REGION Network 5: Клапан регулирующий - 5
   // Зона 7
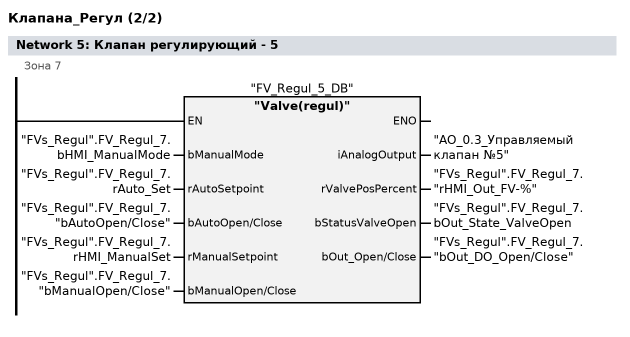
   RUNG wire#powerrail
      "FV_Regul_5_DB"(bManualMode := "FVs_Regul".FV_Regul_7.bHMI_ManualMode, rAutoSetpoint := "FVs_Regul".FV_Regul_7.rAuto_Set, "bAutoOpen/Close" := "FVs_Regul".FV_Regul_7."bAutoOpen/Close", rManualSetpoint := "FVs_Regul".FV_Regul_7.rHMI_ManualSet, "bManualOpen/Close" := "FVs_Regul".FV_Regul_7."bManualOpen/Close", iAnalogOutput => "AO_0.3_Управляемый клапан №5", rValvePosPercent => "FVs_Regul".FV_Regul_7."rHMI_Out_FV-%", bStatusValveOpen => "FVs_Regul".FV_Regul_7.bOut_State_ValveOpen, "bOut_Open/Close" => "FVs_Regul".FV_Regul_7."bOut_DO_Open/Close")
   END_RUNG
   // the same network as SCL:
   "FV_Regul_5_DB"(bManualMode := "FVs_Regul".FV_Regul_7.bHMI_ManualMode,   // "Valve(regul)"
                   rAutoSetpoint := "FVs_Regul".FV_Regul_7.rAuto_Set,
                   "bAutoOpen/Close" := "FVs_Regul".FV_Regul_7."bAutoOpen/Close",
                   rManualSetpoint := "FVs_Regul".FV_Regul_7.rHMI_ManualSet,
                   "bManualOpen/Close" := "FVs_Regul".FV_Regul_7."bManualOpen/Close",
                   iAnalogOutput => "AO_0.3_Управляемый клапан №5",
                   rValvePosPercent => "FVs_Regul".FV_Regul_7."rHMI_Out_FV-%",
                   bStatusValveOpen => "FVs_Regul".FV_Regul_7.bOut_State_ValveOpen,
                   "bOut_Open/Close" => "FVs_Regul".FV_Regul_7."bOut_DO_Open/Close");
END_REGION

REGION Network 6 (SCL): Клапана регулирующие ручной режим с вфходом DO
   // Для перевода клапана регулирующего в ручной режим должен перейти по сигналу от ручного режим с клапана DO, т.е. для работы клапана регулирующего необходим сигнал DO
   (*"FVs_o/p".FV_1.bManualMode := "FVs_Regul".FV_Regul_1.bHMI_ManualMode;
   "FVs_o/p".FV_2.bManualMode := "FVs_Regul".FV_Regul_2.bHMI_ManualMode;
   "FVs_o/p".FV_3.bManualMode := "FVs_Regul".FV_Regul_3.bHMI_ManualMode;
   "FVs_o/p".FV_4.bManualMode := "FVs_Regul".FV_Regul_5.bHMI_ManualMode;
   *)
END_REGION
END_FUNCTION

FUNCTION "Зоны пастеризации_Контроль" : Void   // FC3, LAD
{ S7_Optimized_Access := 'TRUE' }
VERSION : 0.1
BEGIN

REGION Network 1: Зона 1
   // Зона 1
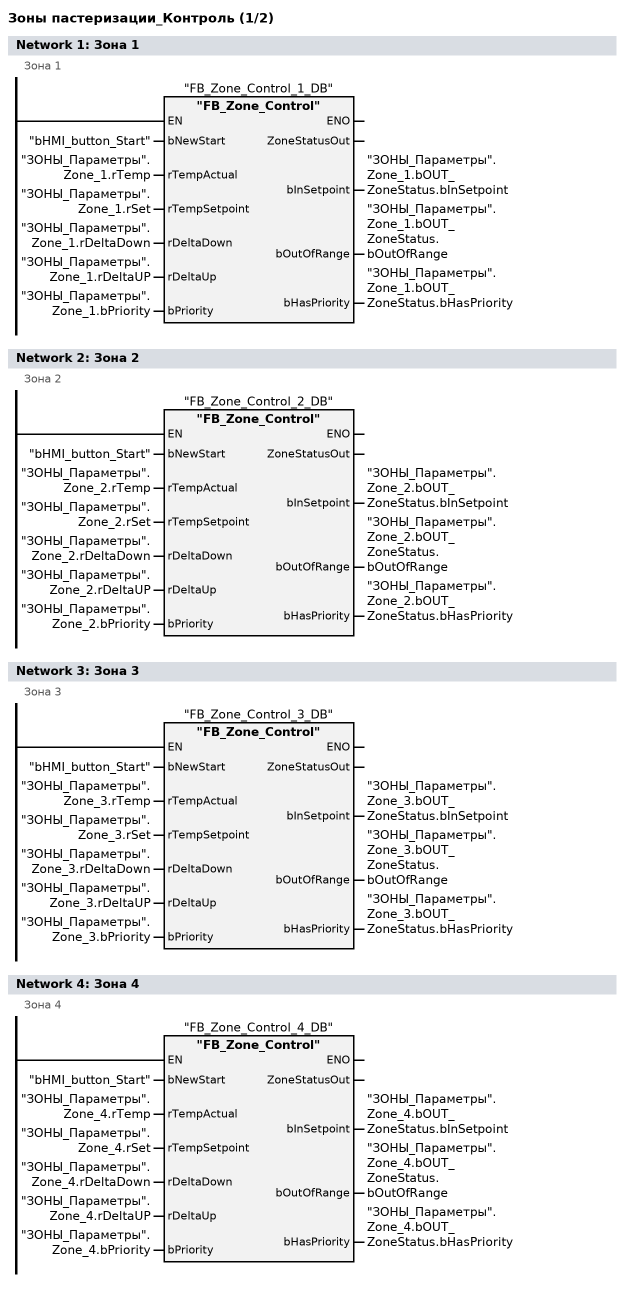
   RUNG wire#powerrail
      "FB_Zone_Control_1_DB"(bNewStart := "bHMI_button_Start", rTempActual := "ЗОНЫ_Параметры".Zone_1.rTemp, rTempSetpoint := "ЗОНЫ_Параметры".Zone_1.rSet, rDeltaDown := "ЗОНЫ_Параметры".Zone_1.rDeltaDown, rDeltaUp := "ЗОНЫ_Параметры".Zone_1.rDeltaUP, bPriority := "ЗОНЫ_Параметры".Zone_1.bPriority, ZoneStatusOut =>, bInSetpoint => "ЗОНЫ_Параметры".Zone_1.bOUT_ZoneStatus.bInSetpoint, bOutOfRange => "ЗОНЫ_Параметры".Zone_1.bOUT_ZoneStatus.bOutOfRange, bHasPriority => "ЗОНЫ_Параметры".Zone_1.bOUT_ZoneStatus.bHasPriority)
   END_RUNG
   // the same network as SCL:
   "FB_Zone_Control_1_DB"(bNewStart := "bHMI_button_Start",   // "FB_Zone_Control"
                          rTempActual := "ЗОНЫ_Параметры".Zone_1.rTemp,
                          rTempSetpoint := "ЗОНЫ_Параметры".Zone_1.rSet,
                          rDeltaDown := "ЗОНЫ_Параметры".Zone_1.rDeltaDown,
                          rDeltaUp := "ЗОНЫ_Параметры".Zone_1.rDeltaUP,
                          bPriority := "ЗОНЫ_Параметры".Zone_1.bPriority,
                          bInSetpoint => "ЗОНЫ_Параметры".Zone_1.bOUT_ZoneStatus.bInSetpoint,
                          bOutOfRange => "ЗОНЫ_Параметры".Zone_1.bOUT_ZoneStatus.bOutOfRange,
                          bHasPriority => "ЗОНЫ_Параметры".Zone_1.bOUT_ZoneStatus.bHasPriority);
END_REGION

REGION Network 2: Зона 2
   // Зона 2
   RUNG wire#powerrail
      "FB_Zone_Control_2_DB"(bNewStart := "bHMI_button_Start", rTempActual := "ЗОНЫ_Параметры".Zone_2.rTemp, rTempSetpoint := "ЗОНЫ_Параметры".Zone_2.rSet, rDeltaDown := "ЗОНЫ_Параметры".Zone_2.rDeltaDown, rDeltaUp := "ЗОНЫ_Параметры".Zone_2.rDeltaUP, bPriority := "ЗОНЫ_Параметры".Zone_2.bPriority, ZoneStatusOut =>, bInSetpoint => "ЗОНЫ_Параметры".Zone_2.bOUT_ZoneStatus.bInSetpoint, bOutOfRange => "ЗОНЫ_Параметры".Zone_2.bOUT_ZoneStatus.bOutOfRange, bHasPriority => "ЗОНЫ_Параметры".Zone_2.bOUT_ZoneStatus.bHasPriority)
   END_RUNG
   // the same network as SCL:
   "FB_Zone_Control_2_DB"(bNewStart := "bHMI_button_Start",   // "FB_Zone_Control"
                          rTempActual := "ЗОНЫ_Параметры".Zone_2.rTemp,
                          rTempSetpoint := "ЗОНЫ_Параметры".Zone_2.rSet,
                          rDeltaDown := "ЗОНЫ_Параметры".Zone_2.rDeltaDown,
                          rDeltaUp := "ЗОНЫ_Параметры".Zone_2.rDeltaUP,
                          bPriority := "ЗОНЫ_Параметры".Zone_2.bPriority,
                          bInSetpoint => "ЗОНЫ_Параметры".Zone_2.bOUT_ZoneStatus.bInSetpoint,
                          bOutOfRange => "ЗОНЫ_Параметры".Zone_2.bOUT_ZoneStatus.bOutOfRange,
                          bHasPriority => "ЗОНЫ_Параметры".Zone_2.bOUT_ZoneStatus.bHasPriority);
END_REGION

REGION Network 3: Зона 3
   // Зона 3
   RUNG wire#powerrail
      "FB_Zone_Control_3_DB"(bNewStart := "bHMI_button_Start", rTempActual := "ЗОНЫ_Параметры".Zone_3.rTemp, rTempSetpoint := "ЗОНЫ_Параметры".Zone_3.rSet, rDeltaDown := "ЗОНЫ_Параметры".Zone_3.rDeltaDown, rDeltaUp := "ЗОНЫ_Параметры".Zone_3.rDeltaUP, bPriority := "ЗОНЫ_Параметры".Zone_3.bPriority, ZoneStatusOut =>, bInSetpoint => "ЗОНЫ_Параметры".Zone_3.bOUT_ZoneStatus.bInSetpoint, bOutOfRange => "ЗОНЫ_Параметры".Zone_3.bOUT_ZoneStatus.bOutOfRange, bHasPriority => "ЗОНЫ_Параметры".Zone_3.bOUT_ZoneStatus.bHasPriority)
   END_RUNG
   // the same network as SCL:
   "FB_Zone_Control_3_DB"(bNewStart := "bHMI_button_Start",   // "FB_Zone_Control"
                          rTempActual := "ЗОНЫ_Параметры".Zone_3.rTemp,
                          rTempSetpoint := "ЗОНЫ_Параметры".Zone_3.rSet,
                          rDeltaDown := "ЗОНЫ_Параметры".Zone_3.rDeltaDown,
                          rDeltaUp := "ЗОНЫ_Параметры".Zone_3.rDeltaUP,
                          bPriority := "ЗОНЫ_Параметры".Zone_3.bPriority,
                          bInSetpoint => "ЗОНЫ_Параметры".Zone_3.bOUT_ZoneStatus.bInSetpoint,
                          bOutOfRange => "ЗОНЫ_Параметры".Zone_3.bOUT_ZoneStatus.bOutOfRange,
                          bHasPriority => "ЗОНЫ_Параметры".Zone_3.bOUT_ZoneStatus.bHasPriority);
END_REGION

REGION Network 4: Зона 4
   // Зона 4
   RUNG wire#powerrail
      "FB_Zone_Control_4_DB"(bNewStart := "bHMI_button_Start", rTempActual := "ЗОНЫ_Параметры".Zone_4.rTemp, rTempSetpoint := "ЗОНЫ_Параметры".Zone_4.rSet, rDeltaDown := "ЗОНЫ_Параметры".Zone_4.rDeltaDown, rDeltaUp := "ЗОНЫ_Параметры".Zone_4.rDeltaUP, bPriority := "ЗОНЫ_Параметры".Zone_4.bPriority, ZoneStatusOut =>, bInSetpoint => "ЗОНЫ_Параметры".Zone_4.bOUT_ZoneStatus.bInSetpoint, bOutOfRange => "ЗОНЫ_Параметры".Zone_4.bOUT_ZoneStatus.bOutOfRange, bHasPriority => "ЗОНЫ_Параметры".Zone_4.bOUT_ZoneStatus.bHasPriority)
   END_RUNG
   // the same network as SCL:
   "FB_Zone_Control_4_DB"(bNewStart := "bHMI_button_Start",   // "FB_Zone_Control"
                          rTempActual := "ЗОНЫ_Параметры".Zone_4.rTemp,
                          rTempSetpoint := "ЗОНЫ_Параметры".Zone_4.rSet,
                          rDeltaDown := "ЗОНЫ_Параметры".Zone_4.rDeltaDown,
                          rDeltaUp := "ЗОНЫ_Параметры".Zone_4.rDeltaUP,
                          bPriority := "ЗОНЫ_Параметры".Zone_4.bPriority,
                          bInSetpoint => "ЗОНЫ_Параметры".Zone_4.bOUT_ZoneStatus.bInSetpoint,
                          bOutOfRange => "ЗОНЫ_Параметры".Zone_4.bOUT_ZoneStatus.bOutOfRange,
                          bHasPriority => "ЗОНЫ_Параметры".Zone_4.bOUT_ZoneStatus.bHasPriority);
END_REGION

REGION Network 5: Зона 5
   // Зона 5
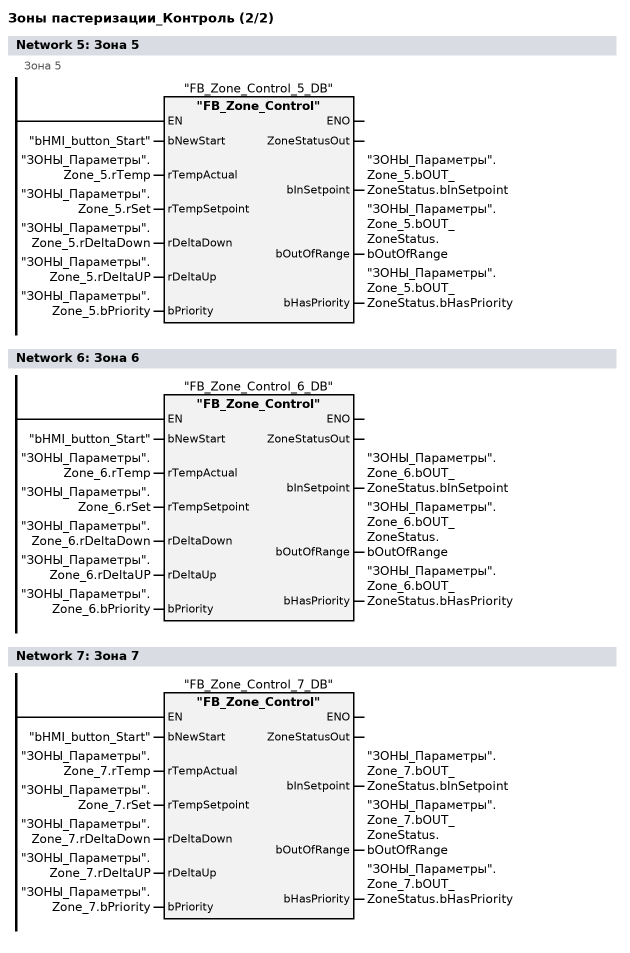
   RUNG wire#powerrail
      "FB_Zone_Control_5_DB"(bNewStart := "bHMI_button_Start", rTempActual := "ЗОНЫ_Параметры".Zone_5.rTemp, rTempSetpoint := "ЗОНЫ_Параметры".Zone_5.rSet, rDeltaDown := "ЗОНЫ_Параметры".Zone_5.rDeltaDown, rDeltaUp := "ЗОНЫ_Параметры".Zone_5.rDeltaUP, bPriority := "ЗОНЫ_Параметры".Zone_5.bPriority, ZoneStatusOut =>, bInSetpoint => "ЗОНЫ_Параметры".Zone_5.bOUT_ZoneStatus.bInSetpoint, bOutOfRange => "ЗОНЫ_Параметры".Zone_5.bOUT_ZoneStatus.bOutOfRange, bHasPriority => "ЗОНЫ_Параметры".Zone_5.bOUT_ZoneStatus.bHasPriority)
   END_RUNG
   // the same network as SCL:
   "FB_Zone_Control_5_DB"(bNewStart := "bHMI_button_Start",   // "FB_Zone_Control"
                          rTempActual := "ЗОНЫ_Параметры".Zone_5.rTemp,
                          rTempSetpoint := "ЗОНЫ_Параметры".Zone_5.rSet,
                          rDeltaDown := "ЗОНЫ_Параметры".Zone_5.rDeltaDown,
                          rDeltaUp := "ЗОНЫ_Параметры".Zone_5.rDeltaUP,
                          bPriority := "ЗОНЫ_Параметры".Zone_5.bPriority,
                          bInSetpoint => "ЗОНЫ_Параметры".Zone_5.bOUT_ZoneStatus.bInSetpoint,
                          bOutOfRange => "ЗОНЫ_Параметры".Zone_5.bOUT_ZoneStatus.bOutOfRange,
                          bHasPriority => "ЗОНЫ_Параметры".Zone_5.bOUT_ZoneStatus.bHasPriority);
END_REGION

REGION Network 6: Зона 6
   RUNG wire#powerrail
      "FB_Zone_Control_6_DB"(bNewStart := "bHMI_button_Start", rTempActual := "ЗОНЫ_Параметры".Zone_6.rTemp, rTempSetpoint := "ЗОНЫ_Параметры".Zone_6.rSet, rDeltaDown := "ЗОНЫ_Параметры".Zone_6.rDeltaDown, rDeltaUp := "ЗОНЫ_Параметры".Zone_6.rDeltaUP, bPriority := "ЗОНЫ_Параметры".Zone_6.bPriority, ZoneStatusOut =>, bInSetpoint => "ЗОНЫ_Параметры".Zone_6.bOUT_ZoneStatus.bInSetpoint, bOutOfRange => "ЗОНЫ_Параметры".Zone_6.bOUT_ZoneStatus.bOutOfRange, bHasPriority => "ЗОНЫ_Параметры".Zone_6.bOUT_ZoneStatus.bHasPriority)
   END_RUNG
   // the same network as SCL:
   "FB_Zone_Control_6_DB"(bNewStart := "bHMI_button_Start",   // "FB_Zone_Control"
                          rTempActual := "ЗОНЫ_Параметры".Zone_6.rTemp,
                          rTempSetpoint := "ЗОНЫ_Параметры".Zone_6.rSet,
                          rDeltaDown := "ЗОНЫ_Параметры".Zone_6.rDeltaDown,
                          rDeltaUp := "ЗОНЫ_Параметры".Zone_6.rDeltaUP,
                          bPriority := "ЗОНЫ_Параметры".Zone_6.bPriority,
                          bInSetpoint => "ЗОНЫ_Параметры".Zone_6.bOUT_ZoneStatus.bInSetpoint,
                          bOutOfRange => "ЗОНЫ_Параметры".Zone_6.bOUT_ZoneStatus.bOutOfRange,
                          bHasPriority => "ЗОНЫ_Параметры".Zone_6.bOUT_ZoneStatus.bHasPriority);
END_REGION

REGION Network 7: Зона 7
   RUNG wire#powerrail
      "FB_Zone_Control_7_DB"(bNewStart := "bHMI_button_Start", rTempActual := "ЗОНЫ_Параметры".Zone_7.rTemp, rTempSetpoint := "ЗОНЫ_Параметры".Zone_7.rSet, rDeltaDown := "ЗОНЫ_Параметры".Zone_7.rDeltaDown, rDeltaUp := "ЗОНЫ_Параметры".Zone_7.rDeltaUP, bPriority := "ЗОНЫ_Параметры".Zone_7.bPriority, ZoneStatusOut =>, bInSetpoint => "ЗОНЫ_Параметры".Zone_7.bOUT_ZoneStatus.bInSetpoint, bOutOfRange => "ЗОНЫ_Параметры".Zone_7.bOUT_ZoneStatus.bOutOfRange, bHasPriority => "ЗОНЫ_Параметры".Zone_7.bOUT_ZoneStatus.bHasPriority)
   END_RUNG
   // the same network as SCL:
   "FB_Zone_Control_7_DB"(bNewStart := "bHMI_button_Start",   // "FB_Zone_Control"
                          rTempActual := "ЗОНЫ_Параметры".Zone_7.rTemp,
                          rTempSetpoint := "ЗОНЫ_Параметры".Zone_7.rSet,
                          rDeltaDown := "ЗОНЫ_Параметры".Zone_7.rDeltaDown,
                          rDeltaUp := "ЗОНЫ_Параметры".Zone_7.rDeltaUP,
                          bPriority := "ЗОНЫ_Параметры".Zone_7.bPriority,
                          bInSetpoint => "ЗОНЫ_Параметры".Zone_7.bOUT_ZoneStatus.bInSetpoint,
                          bOutOfRange => "ЗОНЫ_Параметры".Zone_7.bOUT_ZoneStatus.bOutOfRange,
                          bHasPriority => "ЗОНЫ_Параметры".Zone_7.bOUT_ZoneStatus.bHasPriority);
END_REGION

REGION Network 8 (SCL): Соответствие выхода с датчика температур с входом для темп зоны
   "ЗОНЫ_Параметры".Zone_1.rTemp := "AI_DB".AI_1.rAI_Value;
   "ЗОНЫ_Параметры".Zone_2.rTemp := "AI_DB".AI_2.rAI_Value;
   "ЗОНЫ_Параметры".Zone_3.rTemp := "AI_DB".AI_3.rAI_Value;
   "ЗОНЫ_Параметры".Zone_4.rTemp := "AI_DB".AI_4.rAI_Value;
   "ЗОНЫ_Параметры".Zone_5.rTemp := "AI_DB".AI_5.rAI_Value;
   "ЗОНЫ_Параметры".Zone_6.rTemp := "AI_DB".AI_6.rAI_Value;
   "ЗОНЫ_Параметры".Zone_7.rTemp := "AI_DB".AI_7.rAI_Value;
END_REGION
END_FUNCTION

FUNCTION "Аварии/res" : Void   // FC4, LAD
{ S7_Optimized_Access := 'TRUE' }
VERSION : 0.1
   VAR_INPUT
      bResrt : Bool;
   END_VAR
   VAR_OUTPUT
      xAlarm : Bool;   // Есть активные аварии
   END_VAR
BEGIN

REGION Network 1
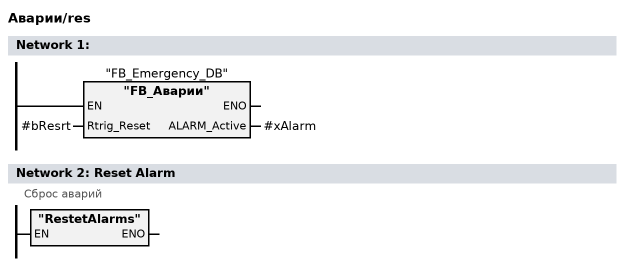
   RUNG wire#powerrail
      "FB_Emergency_DB"(Rtrig_Reset := #bResrt, ALARM_Active => #xAlarm)
   END_RUNG
   // the same network as SCL:
   "FB_Emergency_DB"(Rtrig_Reset := #bResrt, ALARM_Active => #xAlarm);   // "FB_Аварии"
END_REGION

REGION Network 2: Reset Alarm
   // Сброс аварий
   RUNG wire#powerrail
      "RestetAlarms"()
   END_RUNG
   // the same network as SCL:
   "RestetAlarms"();
END_REGION

REGION Network 3 (SCL): Есть активные аварии
END_REGION
END_FUNCTION

FUNCTION "Насосы" : Void   // FC5, LAD
{ S7_Optimized_Access := 'TRUE' }
VERSION : 0.1
// Блоки управления Насосами
BEGIN

REGION Network 1: Насос 1
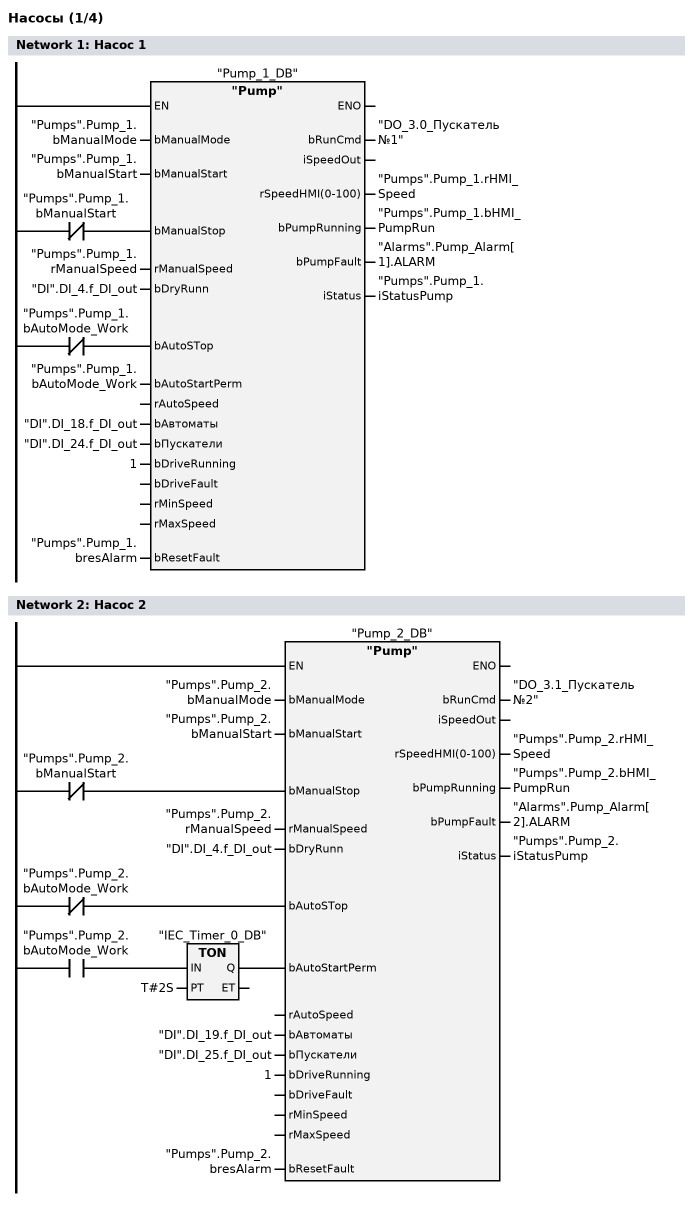
   RUNG wire#powerrail
      "Pump_1_DB"(bManualStop := wire#w1, bAutoSTop := wire#w2, bManualMode := "Pumps".Pump_1.bManualMode, bManualStart := "Pumps".Pump_1.bManualStart, rManualSpeed := "Pumps".Pump_1.rManualSpeed, bDryRunn := "DI".DI_4.f_DI_out, bAutoStartPerm := "Pumps".Pump_1.bAutoMode_Work, rAutoSpeed :=, bАвтоматы := "DI".DI_18.f_DI_out, bПускатели := "DI".DI_24.f_DI_out, bDriveRunning := 1, bDriveFault :=, rMinSpeed :=, rMaxSpeed :=, bResetFault := "Pumps".Pump_1.bresAlarm, bRunCmd => "DO_3.0_Пускатель №1", iSpeedOut =>, "rSpeedHMI(0-100)" => "Pumps".Pump_1.rHMI_Speed, bPumpRunning => "Pumps".Pump_1.bHMI_PumpRun, bPumpFault => "Alarms".Pump_Alarm[1].ALARM, iStatus => "Pumps".Pump_1.iStatusPump)
   END_RUNG
   RUNG wire#powerrail
      I_Contact( "Pumps".Pump_1.bManualStart )
   END_RUNG wire#w1
   RUNG wire#powerrail
      I_Contact( "Pumps".Pump_1.bAutoMode_Work )
   END_RUNG wire#w2
   // the same network as SCL:
   "Pump_1_DB"(bManualMode := "Pumps".Pump_1.bManualMode,   // "Pump"
               bManualStart := "Pumps".Pump_1.bManualStart,
               bManualStop := NOT "Pumps".Pump_1.bManualStart,
               rManualSpeed := "Pumps".Pump_1.rManualSpeed,
               bDryRunn := "DI".DI_4.f_DI_out,
               bAutoSTop := NOT "Pumps".Pump_1.bAutoMode_Work,
               bAutoStartPerm := "Pumps".Pump_1.bAutoMode_Work,
               bАвтоматы := "DI".DI_18.f_DI_out,
               bПускатели := "DI".DI_24.f_DI_out,
               bDriveRunning := 1,
               bResetFault := "Pumps".Pump_1.bresAlarm,
               bRunCmd => "DO_3.0_Пускатель №1",
               "rSpeedHMI(0-100)" => "Pumps".Pump_1.rHMI_Speed,
               bPumpRunning => "Pumps".Pump_1.bHMI_PumpRun,
               bPumpFault => "Alarms".Pump_Alarm[1].ALARM,
               iStatus => "Pumps".Pump_1.iStatusPump);
END_REGION

REGION Network 2: Насос 2
   "IEC_Timer_0_DB".TON(IN := "Pumps".Pump_2.bAutoMode_Work, PT := T#2S);
   "Pump_2_DB"(bManualMode := "Pumps".Pump_2.bManualMode,   // "Pump"
               bManualStart := "Pumps".Pump_2.bManualStart,
               bManualStop := NOT "Pumps".Pump_2.bManualStart,
               rManualSpeed := "Pumps".Pump_2.rManualSpeed,
               bDryRunn := "DI".DI_4.f_DI_out,
               bAutoSTop := NOT "Pumps".Pump_2.bAutoMode_Work,
               bAutoStartPerm := "IEC_Timer_0_DB".Q,
               bАвтоматы := "DI".DI_19.f_DI_out,
               bПускатели := "DI".DI_25.f_DI_out,
               bDriveRunning := 1,
               bResetFault := "Pumps".Pump_2.bresAlarm,
               bRunCmd => "DO_3.1_Пускатель №2",
               "rSpeedHMI(0-100)" => "Pumps".Pump_2.rHMI_Speed,
               bPumpRunning => "Pumps".Pump_2.bHMI_PumpRun,
               bPumpFault => "Alarms".Pump_Alarm[2].ALARM,
               iStatus => "Pumps".Pump_2.iStatusPump);
END_REGION

REGION Network 3: Насос 3
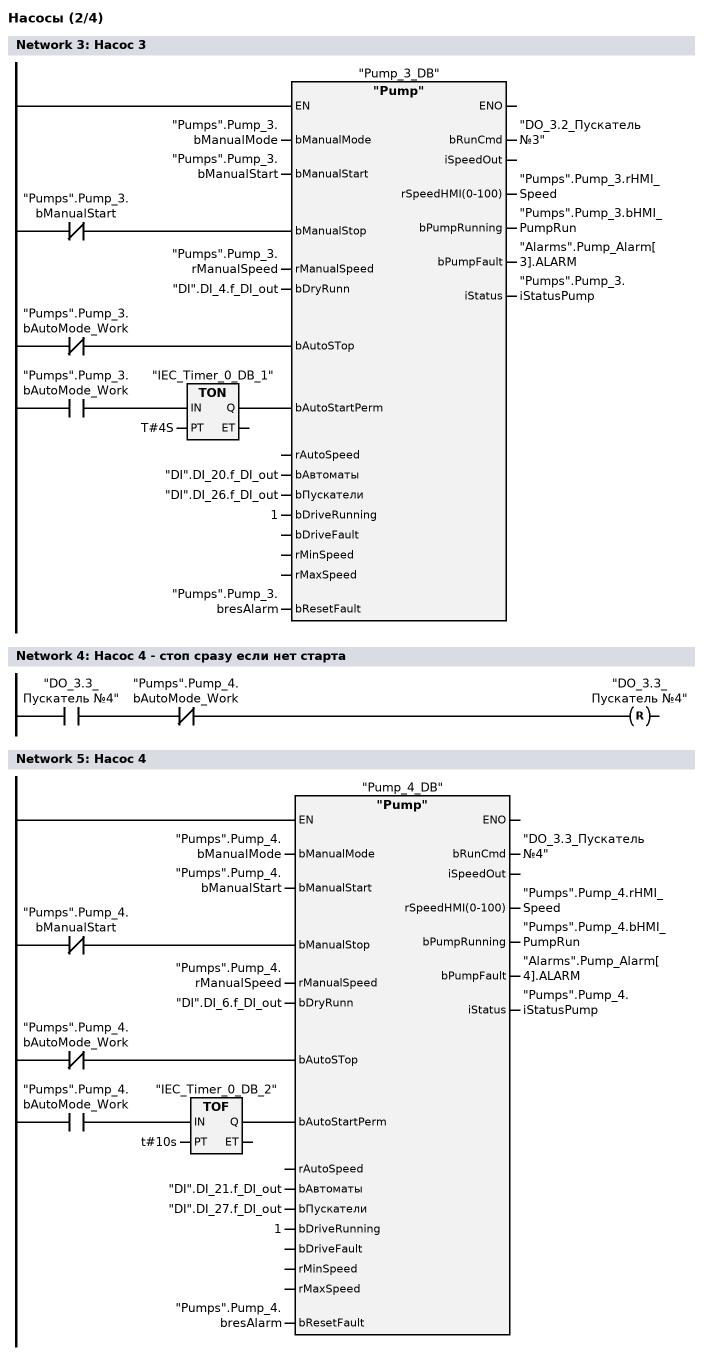
   "IEC_Timer_0_DB_1".TON(IN := "Pumps".Pump_3.bAutoMode_Work, PT := T#4S);
   "Pump_3_DB"(bManualMode := "Pumps".Pump_3.bManualMode,   // "Pump"
               bManualStart := "Pumps".Pump_3.bManualStart,
               bManualStop := NOT "Pumps".Pump_3.bManualStart,
               rManualSpeed := "Pumps".Pump_3.rManualSpeed,
               bDryRunn := "DI".DI_4.f_DI_out,
               bAutoSTop := NOT "Pumps".Pump_3.bAutoMode_Work,
               bAutoStartPerm := "IEC_Timer_0_DB_1".Q,
               bАвтоматы := "DI".DI_20.f_DI_out,
               bПускатели := "DI".DI_26.f_DI_out,
               bDriveRunning := 1,
               bResetFault := "Pumps".Pump_3.bresAlarm,
               bRunCmd => "DO_3.2_Пускатель №3",
               "rSpeedHMI(0-100)" => "Pumps".Pump_3.rHMI_Speed,
               bPumpRunning => "Pumps".Pump_3.bHMI_PumpRun,
               bPumpFault => "Alarms".Pump_Alarm[3].ALARM,
               iStatus => "Pumps".Pump_3.iStatusPump);
END_REGION

REGION Network 4: Насос 4 - стоп сразу если нет старта
   RUNG wire#powerrail
      Contact( "DO_3.3_Пускатель №4" )
      I_Contact( "Pumps".Pump_4.bAutoMode_Work )
      R_Coil( "DO_3.3_Пускатель №4" )
   END_RUNG
   // the same network as SCL:
   IF "DO_3.3_Пускатель №4" AND NOT "Pumps".Pump_4.bAutoMode_Work THEN
       "DO_3.3_Пускатель №4" := FALSE;
   END_IF;
END_REGION

REGION Network 5: Насос 4
   "IEC_Timer_0_DB_2".TOF(IN := "Pumps".Pump_4.bAutoMode_Work, PT := t#10s);
   "Pump_4_DB"(bManualMode := "Pumps".Pump_4.bManualMode,   // "Pump"
               bManualStart := "Pumps".Pump_4.bManualStart,
               bManualStop := NOT "Pumps".Pump_4.bManualStart,
               rManualSpeed := "Pumps".Pump_4.rManualSpeed,
               bDryRunn := "DI".DI_6.f_DI_out,
               bAutoSTop := NOT "Pumps".Pump_4.bAutoMode_Work,
               bAutoStartPerm := "IEC_Timer_0_DB_2".Q,
               bАвтоматы := "DI".DI_21.f_DI_out,
               bПускатели := "DI".DI_27.f_DI_out,
               bDriveRunning := 1,
               bResetFault := "Pumps".Pump_4.bresAlarm,
               bRunCmd => "DO_3.3_Пускатель №4",
               "rSpeedHMI(0-100)" => "Pumps".Pump_4.rHMI_Speed,
               bPumpRunning => "Pumps".Pump_4.bHMI_PumpRun,
               bPumpFault => "Alarms".Pump_Alarm[4].ALARM,
               iStatus => "Pumps".Pump_4.iStatusPump);
END_REGION

REGION Network 6: Насос 5
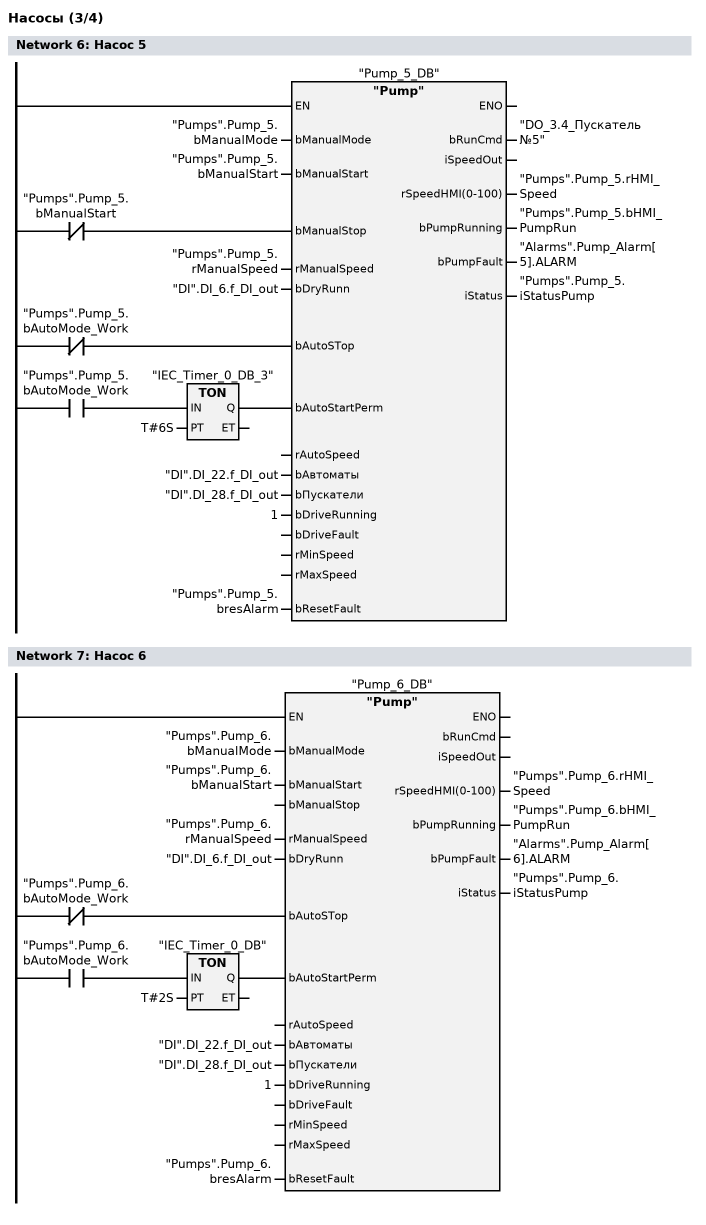
   "IEC_Timer_0_DB_3".TON(IN := "Pumps".Pump_5.bAutoMode_Work, PT := T#6S);
   "Pump_5_DB"(bManualMode := "Pumps".Pump_5.bManualMode,   // "Pump"
               bManualStart := "Pumps".Pump_5.bManualStart,
               bManualStop := NOT "Pumps".Pump_5.bManualStart,
               rManualSpeed := "Pumps".Pump_5.rManualSpeed,
               bDryRunn := "DI".DI_6.f_DI_out,
               bAutoSTop := NOT "Pumps".Pump_5.bAutoMode_Work,
               bAutoStartPerm := "IEC_Timer_0_DB_3".Q,
               bАвтоматы := "DI".DI_22.f_DI_out,
               bПускатели := "DI".DI_28.f_DI_out,
               bDriveRunning := 1,
               bResetFault := "Pumps".Pump_5.bresAlarm,
               bRunCmd => "DO_3.4_Пускатель №5",
               "rSpeedHMI(0-100)" => "Pumps".Pump_5.rHMI_Speed,
               bPumpRunning => "Pumps".Pump_5.bHMI_PumpRun,
               bPumpFault => "Alarms".Pump_Alarm[5].ALARM,
               iStatus => "Pumps".Pump_5.iStatusPump);
END_REGION

REGION Network 7: Насос 6
   "IEC_Timer_0_DB".TON(IN := "Pumps".Pump_6.bAutoMode_Work, PT := T#2S);
   "Pump_6_DB"(bManualMode := "Pumps".Pump_6.bManualMode,   // "Pump"
               bManualStart := "Pumps".Pump_6.bManualStart,
               rManualSpeed := "Pumps".Pump_6.rManualSpeed,
               bDryRunn := "DI".DI_6.f_DI_out,
               bAutoSTop := NOT "Pumps".Pump_6.bAutoMode_Work,
               bAutoStartPerm := "IEC_Timer_0_DB".Q,
               bАвтоматы := "DI".DI_22.f_DI_out,
               bПускатели := "DI".DI_28.f_DI_out,
               bDriveRunning := 1,
               bResetFault := "Pumps".Pump_6.bresAlarm,
               "rSpeedHMI(0-100)" => "Pumps".Pump_6.rHMI_Speed,
               bPumpRunning => "Pumps".Pump_6.bHMI_PumpRun,
               bPumpFault => "Alarms".Pump_Alarm[6].ALARM,
               iStatus => "Pumps".Pump_6.iStatusPump);
END_REGION

REGION Network 8: Насос 7
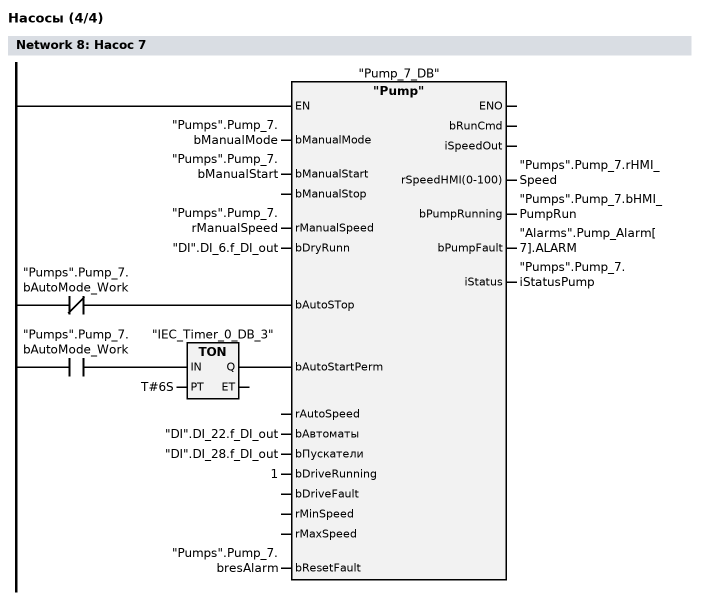
   "IEC_Timer_0_DB_3".TON(IN := "Pumps".Pump_7.bAutoMode_Work, PT := T#6S);
   "Pump_7_DB"(bManualMode := "Pumps".Pump_7.bManualMode,   // "Pump"
               bManualStart := "Pumps".Pump_7.bManualStart,
               rManualSpeed := "Pumps".Pump_7.rManualSpeed,
               bDryRunn := "DI".DI_6.f_DI_out,
               bAutoSTop := NOT "Pumps".Pump_7.bAutoMode_Work,
               bAutoStartPerm := "IEC_Timer_0_DB_3".Q,
               bАвтоматы := "DI".DI_22.f_DI_out,
               bПускатели := "DI".DI_28.f_DI_out,
               bDriveRunning := 1,
               bResetFault := "Pumps".Pump_7.bresAlarm,
               "rSpeedHMI(0-100)" => "Pumps".Pump_7.rHMI_Speed,
               bPumpRunning => "Pumps".Pump_7.bHMI_PumpRun,
               bPumpFault => "Alarms".Pump_Alarm[7].ALARM,
               iStatus => "Pumps".Pump_7.iStatusPump);
END_REGION
END_FUNCTION

FUNCTION "Analogs_IN_All" : Void   // FC6, LAD
TITLE = Датчики AI
{ S7_Optimized_Access := 'FALSE' }
VERSION : 0.1
// Темп - PT100 - 5 шт
// Давление 4-20 - 3 шт
BEGIN

REGION Network 1: Датчик температуры - 1
   // РТ-100
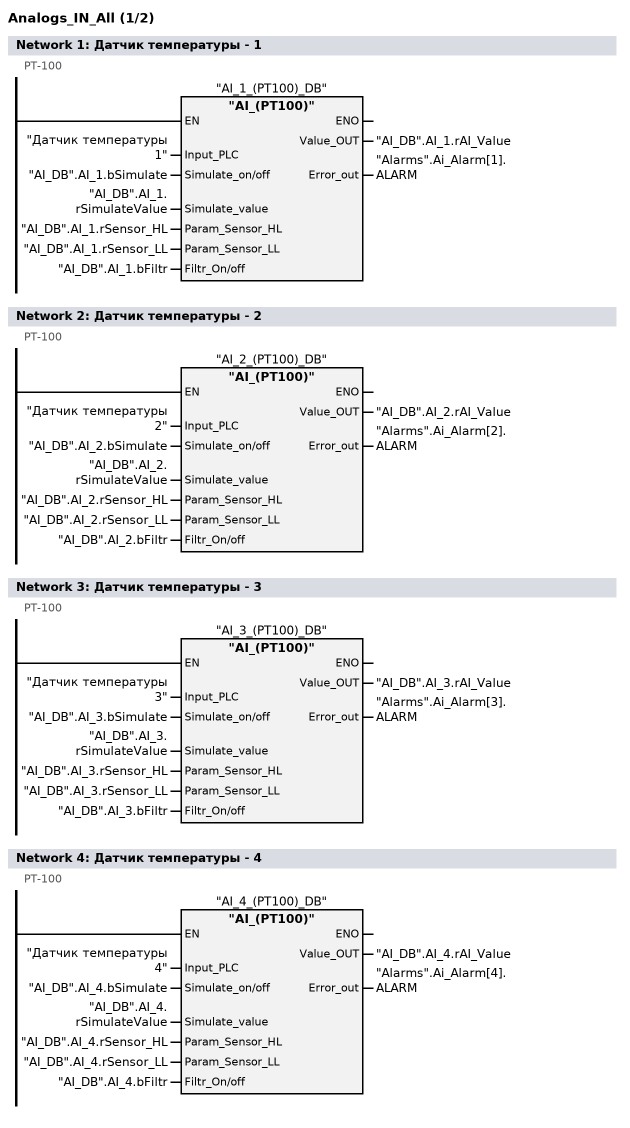
   RUNG wire#powerrail
      "AI_1_(PT100)_DB"(Input_PLC := "Датчик температуры 1", "Simulate_on/off" := "AI_DB".AI_1.bSimulate, Simulate_value := "AI_DB".AI_1.rSimulateValue, Param_Sensor_HL := "AI_DB".AI_1.rSensor_HL, Param_Sensor_LL := "AI_DB".AI_1.rSensor_LL, "Filtr_On/off" := "AI_DB".AI_1.bFiltr, Value_OUT => "AI_DB".AI_1.rAI_Value, Error_out => "Alarms".Ai_Alarm[1].ALARM)
   END_RUNG
   // the same network as SCL:
   "AI_1_(PT100)_DB"(Input_PLC := "Датчик температуры 1",   // "AI_(PT100)"
                     "Simulate_on/off" := "AI_DB".AI_1.bSimulate,
                     Simulate_value := "AI_DB".AI_1.rSimulateValue,
                     Param_Sensor_HL := "AI_DB".AI_1.rSensor_HL,
                     Param_Sensor_LL := "AI_DB".AI_1.rSensor_LL,
                     "Filtr_On/off" := "AI_DB".AI_1.bFiltr,
                     Value_OUT => "AI_DB".AI_1.rAI_Value,
                     Error_out => "Alarms".Ai_Alarm[1].ALARM);
END_REGION

REGION Network 2: Датчик температуры - 2
   // РТ-100
   RUNG wire#powerrail
      "AI_2_(PT100)_DB"(Input_PLC := "Датчик температуры 2", "Simulate_on/off" := "AI_DB".AI_2.bSimulate, Simulate_value := "AI_DB".AI_2.rSimulateValue, Param_Sensor_HL := "AI_DB".AI_2.rSensor_HL, Param_Sensor_LL := "AI_DB".AI_2.rSensor_LL, "Filtr_On/off" := "AI_DB".AI_2.bFiltr, Value_OUT => "AI_DB".AI_2.rAI_Value, Error_out => "Alarms".Ai_Alarm[2].ALARM)
   END_RUNG
   // the same network as SCL:
   "AI_2_(PT100)_DB"(Input_PLC := "Датчик температуры 2",   // "AI_(PT100)"
                     "Simulate_on/off" := "AI_DB".AI_2.bSimulate,
                     Simulate_value := "AI_DB".AI_2.rSimulateValue,
                     Param_Sensor_HL := "AI_DB".AI_2.rSensor_HL,
                     Param_Sensor_LL := "AI_DB".AI_2.rSensor_LL,
                     "Filtr_On/off" := "AI_DB".AI_2.bFiltr,
                     Value_OUT => "AI_DB".AI_2.rAI_Value,
                     Error_out => "Alarms".Ai_Alarm[2].ALARM);
END_REGION

REGION Network 3: Датчик температуры - 3
   // РТ-100
   RUNG wire#powerrail
      "AI_3_(PT100)_DB"(Input_PLC := "Датчик температуры 3", "Simulate_on/off" := "AI_DB".AI_3.bSimulate, Simulate_value := "AI_DB".AI_3.rSimulateValue, Param_Sensor_HL := "AI_DB".AI_3.rSensor_HL, Param_Sensor_LL := "AI_DB".AI_3.rSensor_LL, "Filtr_On/off" := "AI_DB".AI_3.bFiltr, Value_OUT => "AI_DB".AI_3.rAI_Value, Error_out => "Alarms".Ai_Alarm[3].ALARM)
   END_RUNG
   // the same network as SCL:
   "AI_3_(PT100)_DB"(Input_PLC := "Датчик температуры 3",   // "AI_(PT100)"
                     "Simulate_on/off" := "AI_DB".AI_3.bSimulate,
                     Simulate_value := "AI_DB".AI_3.rSimulateValue,
                     Param_Sensor_HL := "AI_DB".AI_3.rSensor_HL,
                     Param_Sensor_LL := "AI_DB".AI_3.rSensor_LL,
                     "Filtr_On/off" := "AI_DB".AI_3.bFiltr,
                     Value_OUT => "AI_DB".AI_3.rAI_Value,
                     Error_out => "Alarms".Ai_Alarm[3].ALARM);
END_REGION

REGION Network 4: Датчик температуры - 4
   // РТ-100
   RUNG wire#powerrail
      "AI_4_(PT100)_DB"(Input_PLC := "Датчик температуры 4", "Simulate_on/off" := "AI_DB".AI_4.bSimulate, Simulate_value := "AI_DB".AI_4.rSimulateValue, Param_Sensor_HL := "AI_DB".AI_4.rSensor_HL, Param_Sensor_LL := "AI_DB".AI_4.rSensor_LL, "Filtr_On/off" := "AI_DB".AI_4.bFiltr, Value_OUT => "AI_DB".AI_4.rAI_Value, Error_out => "Alarms".Ai_Alarm[4].ALARM)
   END_RUNG
   // the same network as SCL:
   "AI_4_(PT100)_DB"(Input_PLC := "Датчик температуры 4",   // "AI_(PT100)"
                     "Simulate_on/off" := "AI_DB".AI_4.bSimulate,
                     Simulate_value := "AI_DB".AI_4.rSimulateValue,
                     Param_Sensor_HL := "AI_DB".AI_4.rSensor_HL,
                     Param_Sensor_LL := "AI_DB".AI_4.rSensor_LL,
                     "Filtr_On/off" := "AI_DB".AI_4.bFiltr,
                     Value_OUT => "AI_DB".AI_4.rAI_Value,
                     Error_out => "Alarms".Ai_Alarm[4].ALARM);
END_REGION

REGION Network 5: Датчик температуры - 5
   // РТ-100
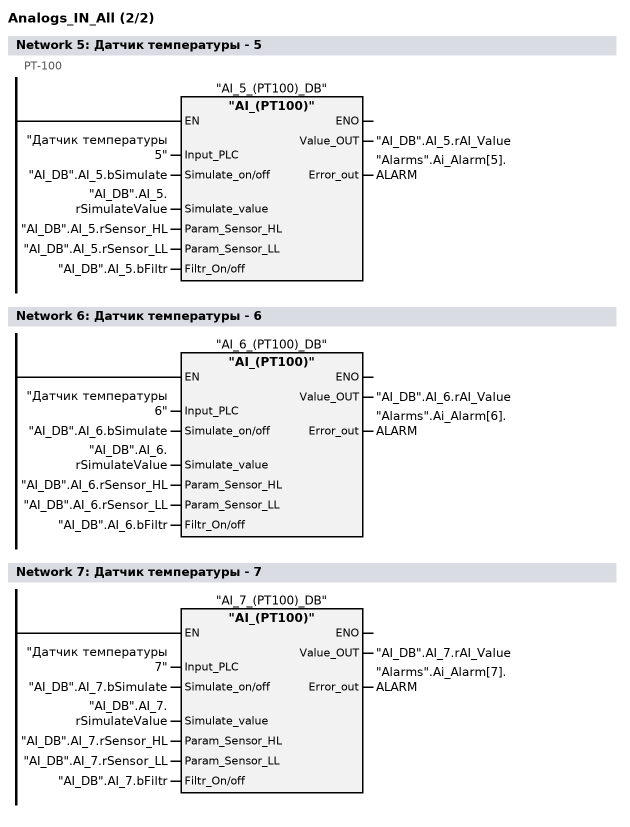
   RUNG wire#powerrail
      "AI_5_(PT100)_DB"(Input_PLC := "Датчик температуры 5", "Simulate_on/off" := "AI_DB".AI_5.bSimulate, Simulate_value := "AI_DB".AI_5.rSimulateValue, Param_Sensor_HL := "AI_DB".AI_5.rSensor_HL, Param_Sensor_LL := "AI_DB".AI_5.rSensor_LL, "Filtr_On/off" := "AI_DB".AI_5.bFiltr, Value_OUT => "AI_DB".AI_5.rAI_Value, Error_out => "Alarms".Ai_Alarm[5].ALARM)
   END_RUNG
   // the same network as SCL:
   "AI_5_(PT100)_DB"(Input_PLC := "Датчик температуры 5",   // "AI_(PT100)"
                     "Simulate_on/off" := "AI_DB".AI_5.bSimulate,
                     Simulate_value := "AI_DB".AI_5.rSimulateValue,
                     Param_Sensor_HL := "AI_DB".AI_5.rSensor_HL,
                     Param_Sensor_LL := "AI_DB".AI_5.rSensor_LL,
                     "Filtr_On/off" := "AI_DB".AI_5.bFiltr,
                     Value_OUT => "AI_DB".AI_5.rAI_Value,
                     Error_out => "Alarms".Ai_Alarm[5].ALARM);
END_REGION

REGION Network 6: Датчик температуры - 6
   RUNG wire#powerrail
      "AI_6_(PT100)_DB"(Input_PLC := "Датчик температуры 6", "Simulate_on/off" := "AI_DB".AI_6.bSimulate, Simulate_value := "AI_DB".AI_6.rSimulateValue, Param_Sensor_HL := "AI_DB".AI_6.rSensor_HL, Param_Sensor_LL := "AI_DB".AI_6.rSensor_LL, "Filtr_On/off" := "AI_DB".AI_6.bFiltr, Value_OUT => "AI_DB".AI_6.rAI_Value, Error_out => "Alarms".Ai_Alarm[6].ALARM)
   END_RUNG
   // the same network as SCL:
   "AI_6_(PT100)_DB"(Input_PLC := "Датчик температуры 6",   // "AI_(PT100)"
                     "Simulate_on/off" := "AI_DB".AI_6.bSimulate,
                     Simulate_value := "AI_DB".AI_6.rSimulateValue,
                     Param_Sensor_HL := "AI_DB".AI_6.rSensor_HL,
                     Param_Sensor_LL := "AI_DB".AI_6.rSensor_LL,
                     "Filtr_On/off" := "AI_DB".AI_6.bFiltr,
                     Value_OUT => "AI_DB".AI_6.rAI_Value,
                     Error_out => "Alarms".Ai_Alarm[6].ALARM);
END_REGION

REGION Network 7: Датчик температуры - 7
   RUNG wire#powerrail
      "AI_7_(PT100)_DB"(Input_PLC := "Датчик температуры 7", "Simulate_on/off" := "AI_DB".AI_7.bSimulate, Simulate_value := "AI_DB".AI_7.rSimulateValue, Param_Sensor_HL := "AI_DB".AI_7.rSensor_HL, Param_Sensor_LL := "AI_DB".AI_7.rSensor_LL, "Filtr_On/off" := "AI_DB".AI_7.bFiltr, Value_OUT => "AI_DB".AI_7.rAI_Value, Error_out => "Alarms".Ai_Alarm[7].ALARM)
   END_RUNG
   // the same network as SCL:
   "AI_7_(PT100)_DB"(Input_PLC := "Датчик температуры 7",   // "AI_(PT100)"
                     "Simulate_on/off" := "AI_DB".AI_7.bSimulate,
                     Simulate_value := "AI_DB".AI_7.rSimulateValue,
                     Param_Sensor_HL := "AI_DB".AI_7.rSensor_HL,
                     Param_Sensor_LL := "AI_DB".AI_7.rSensor_LL,
                     "Filtr_On/off" := "AI_DB".AI_7.bFiltr,
                     Value_OUT => "AI_DB".AI_7.rAI_Value,
                     Error_out => "Alarms".Ai_Alarm[7].ALARM);
END_REGION
END_FUNCTION

FUNCTION "Discret_Inputs_All" : Void   // FC8, LAD
TITLE = Для сбора всех DI в одном месте
{ S7_Optimized_Access := 'FALSE' }
VERSION : 0.1
   VAR CONSTANT
      Cons_TimeDelay : DInt := 100;
   END_VAR
BEGIN

REGION Network 1: E-Stop1
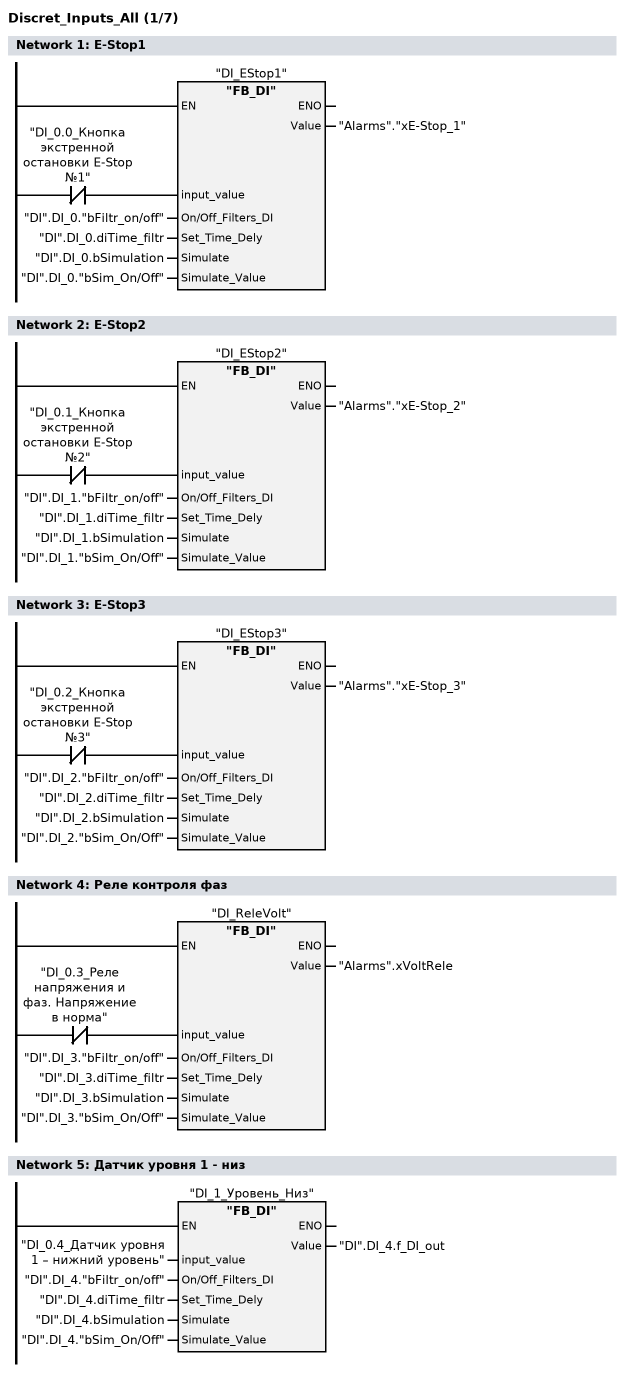
   RUNG wire#powerrail
      "DI_EStop1"(input_value := wire#w1, "On/Off_Filters_DI" := "DI".DI_0."bFiltr_on/off", Set_Time_Dely := "DI".DI_0.diTime_filtr, Simulate := "DI".DI_0.bSimulation, Simulate_Value := "DI".DI_0."bSim_On/Off", Value => "Alarms"."xE-Stop_1")
   END_RUNG
   RUNG wire#powerrail
      I_Contact( "DI_0.0_Кнопка экстренной остановки E-Stop №1" )
   END_RUNG wire#w1
   // the same network as SCL:
   "DI_EStop1"(input_value := NOT "DI_0.0_Кнопка экстренной остановки E-Stop №1",   // "FB_DI"
               "On/Off_Filters_DI" := "DI".DI_0."bFiltr_on/off",
               Set_Time_Dely := "DI".DI_0.diTime_filtr,
               Simulate := "DI".DI_0.bSimulation,
               Simulate_Value := "DI".DI_0."bSim_On/Off",
               Value => "Alarms"."xE-Stop_1");
END_REGION

REGION Network 2: E-Stop2
   RUNG wire#powerrail
      "DI_EStop2"(input_value := wire#w1, "On/Off_Filters_DI" := "DI".DI_1."bFiltr_on/off", Set_Time_Dely := "DI".DI_1.diTime_filtr, Simulate := "DI".DI_1.bSimulation, Simulate_Value := "DI".DI_1."bSim_On/Off", Value => "Alarms"."xE-Stop_2")
   END_RUNG
   RUNG wire#powerrail
      I_Contact( "DI_0.1_Кнопка экстренной остановки E-Stop №2" )
   END_RUNG wire#w1
   // the same network as SCL:
   "DI_EStop2"(input_value := NOT "DI_0.1_Кнопка экстренной остановки E-Stop №2",   // "FB_DI"
               "On/Off_Filters_DI" := "DI".DI_1."bFiltr_on/off",
               Set_Time_Dely := "DI".DI_1.diTime_filtr,
               Simulate := "DI".DI_1.bSimulation,
               Simulate_Value := "DI".DI_1."bSim_On/Off",
               Value => "Alarms"."xE-Stop_2");
END_REGION

REGION Network 3: E-Stop3
   RUNG wire#powerrail
      "DI_EStop3"(input_value := wire#w1, "On/Off_Filters_DI" := "DI".DI_2."bFiltr_on/off", Set_Time_Dely := "DI".DI_2.diTime_filtr, Simulate := "DI".DI_2.bSimulation, Simulate_Value := "DI".DI_2."bSim_On/Off", Value => "Alarms"."xE-Stop_3")
   END_RUNG
   RUNG wire#powerrail
      I_Contact( "DI_0.2_Кнопка экстренной остановки E-Stop №3" )
   END_RUNG wire#w1
   // the same network as SCL:
   "DI_EStop3"(input_value := NOT "DI_0.2_Кнопка экстренной остановки E-Stop №3",   // "FB_DI"
               "On/Off_Filters_DI" := "DI".DI_2."bFiltr_on/off",
               Set_Time_Dely := "DI".DI_2.diTime_filtr,
               Simulate := "DI".DI_2.bSimulation,
               Simulate_Value := "DI".DI_2."bSim_On/Off",
               Value => "Alarms"."xE-Stop_3");
END_REGION

REGION Network 4: Реле контроля фаз
   RUNG wire#powerrail
      "DI_ReleVolt"(input_value := wire#w1, "On/Off_Filters_DI" := "DI".DI_3."bFiltr_on/off", Set_Time_Dely := "DI".DI_3.diTime_filtr, Simulate := "DI".DI_3.bSimulation, Simulate_Value := "DI".DI_3."bSim_On/Off", Value => "Alarms".xVoltRele)
   END_RUNG
   RUNG wire#powerrail
      I_Contact( "DI_0.3_Реле напряжения и фаз. Напряжение в норма" )
   END_RUNG wire#w1
   // the same network as SCL:
   "DI_ReleVolt"(input_value := NOT "DI_0.3_Реле напряжения и фаз. Напряжение в норма",   // "FB_DI"
                 "On/Off_Filters_DI" := "DI".DI_3."bFiltr_on/off",
                 Set_Time_Dely := "DI".DI_3.diTime_filtr,
                 Simulate := "DI".DI_3.bSimulation,
                 Simulate_Value := "DI".DI_3."bSim_On/Off",
                 Value => "Alarms".xVoltRele);
END_REGION

REGION Network 5: Датчик уровня 1 - низ
   RUNG wire#powerrail
      "DI_1_Уровень_Низ"(input_value := "DI_0.4_Датчик уровня 1 – нижний уровень", "On/Off_Filters_DI" := "DI".DI_4."bFiltr_on/off", Set_Time_Dely := "DI".DI_4.diTime_filtr, Simulate := "DI".DI_4.bSimulation, Simulate_Value := "DI".DI_4."bSim_On/Off", Value => "DI".DI_4.f_DI_out)
   END_RUNG
   // the same network as SCL:
   "DI_1_Уровень_Низ"(input_value := "DI_0.4_Датчик уровня 1 – нижний уровень",   // "FB_DI"
                      "On/Off_Filters_DI" := "DI".DI_4."bFiltr_on/off",
                      Set_Time_Dely := "DI".DI_4.diTime_filtr,
                      Simulate := "DI".DI_4.bSimulation,
                      Simulate_Value := "DI".DI_4."bSim_On/Off",
                      Value => "DI".DI_4.f_DI_out);
END_REGION

REGION Network 6: Датчик уровня 1 - Верх
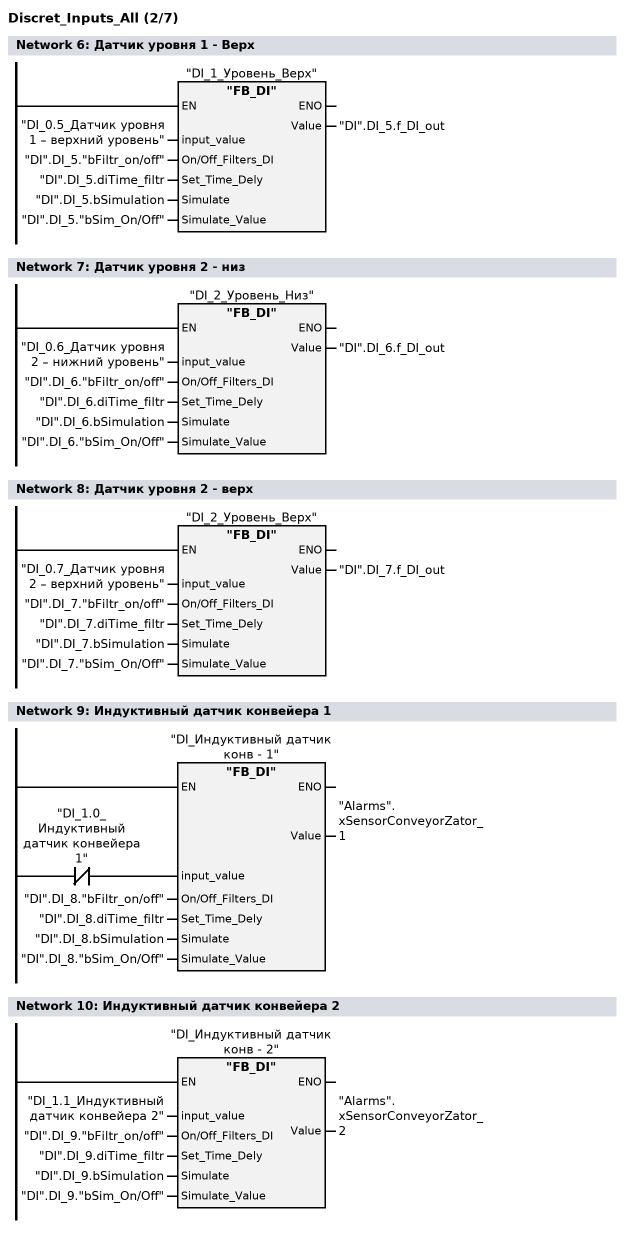
   RUNG wire#powerrail
      "DI_1_Уровень_Верх"(input_value := "DI_0.5_Датчик уровня 1 – верхний уровень", "On/Off_Filters_DI" := "DI".DI_5."bFiltr_on/off", Set_Time_Dely := "DI".DI_5.diTime_filtr, Simulate := "DI".DI_5.bSimulation, Simulate_Value := "DI".DI_5."bSim_On/Off", Value => "DI".DI_5.f_DI_out)
   END_RUNG
   // the same network as SCL:
   "DI_1_Уровень_Верх"(input_value := "DI_0.5_Датчик уровня 1 – верхний уровень",   // "FB_DI"
                       "On/Off_Filters_DI" := "DI".DI_5."bFiltr_on/off",
                       Set_Time_Dely := "DI".DI_5.diTime_filtr,
                       Simulate := "DI".DI_5.bSimulation,
                       Simulate_Value := "DI".DI_5."bSim_On/Off",
                       Value => "DI".DI_5.f_DI_out);
END_REGION

REGION Network 7: Датчик уровня 2 - низ
   RUNG wire#powerrail
      "DI_2_Уровень_Низ"(input_value := "DI_0.6_Датчик уровня 2 – нижний уровень", "On/Off_Filters_DI" := "DI".DI_6."bFiltr_on/off", Set_Time_Dely := "DI".DI_6.diTime_filtr, Simulate := "DI".DI_6.bSimulation, Simulate_Value := "DI".DI_6."bSim_On/Off", Value => "DI".DI_6.f_DI_out)
   END_RUNG
   // the same network as SCL:
   "DI_2_Уровень_Низ"(input_value := "DI_0.6_Датчик уровня 2 – нижний уровень",   // "FB_DI"
                      "On/Off_Filters_DI" := "DI".DI_6."bFiltr_on/off",
                      Set_Time_Dely := "DI".DI_6.diTime_filtr,
                      Simulate := "DI".DI_6.bSimulation,
                      Simulate_Value := "DI".DI_6."bSim_On/Off",
                      Value => "DI".DI_6.f_DI_out);
END_REGION

REGION Network 8: Датчик уровня 2 - верх
   RUNG wire#powerrail
      "DI_2_Уровень_Верх"(input_value := "DI_0.7_Датчик уровня 2 – верхний уровень", "On/Off_Filters_DI" := "DI".DI_7."bFiltr_on/off", Set_Time_Dely := "DI".DI_7.diTime_filtr, Simulate := "DI".DI_7.bSimulation, Simulate_Value := "DI".DI_7."bSim_On/Off", Value => "DI".DI_7.f_DI_out)
   END_RUNG
   // the same network as SCL:
   "DI_2_Уровень_Верх"(input_value := "DI_0.7_Датчик уровня 2 – верхний уровень",   // "FB_DI"
                       "On/Off_Filters_DI" := "DI".DI_7."bFiltr_on/off",
                       Set_Time_Dely := "DI".DI_7.diTime_filtr,
                       Simulate := "DI".DI_7.bSimulation,
                       Simulate_Value := "DI".DI_7."bSim_On/Off",
                       Value => "DI".DI_7.f_DI_out);
END_REGION

REGION Network 9: Индуктивный датчик конвейера 1
   RUNG wire#powerrail
      "DI_Индуктивный датчик конв - 1"(input_value := wire#w1, "On/Off_Filters_DI" := "DI".DI_8."bFiltr_on/off", Set_Time_Dely := "DI".DI_8.diTime_filtr, Simulate := "DI".DI_8.bSimulation, Simulate_Value := "DI".DI_8."bSim_On/Off", Value => "Alarms".xSensorConveyorZator_1)
   END_RUNG
   RUNG wire#powerrail
      I_Contact( "DI_1.0_Индуктивный датчик конвейера 1" )
   END_RUNG wire#w1
   // the same network as SCL:
   "DI_Индуктивный датчик конв - 1"(input_value := NOT "DI_1.0_Индуктивный датчик конвейера 1",   // "FB_DI"
                           "On/Off_Filters_DI" := "DI".DI_8."bFiltr_on/off",
                           Set_Time_Dely := "DI".DI_8.diTime_filtr,
                           Simulate := "DI".DI_8.bSimulation,
                           Simulate_Value := "DI".DI_8."bSim_On/Off",
                           Value => "Alarms".xSensorConveyorZator_1);
END_REGION

REGION Network 10: Индуктивный датчик конвейера 2
   RUNG wire#powerrail
      "DI_Индуктивный датчик конв - 2"(input_value := "DI_1.1_Индуктивный датчик конвейера 2", "On/Off_Filters_DI" := "DI".DI_9."bFiltr_on/off", Set_Time_Dely := "DI".DI_9.diTime_filtr, Simulate := "DI".DI_9.bSimulation, Simulate_Value := "DI".DI_9."bSim_On/Off", Value => "Alarms".xSensorConveyorZator_2)
   END_RUNG
   // the same network as SCL:
   "DI_Индуктивный датчик конв - 2"(input_value := "DI_1.1_Индуктивный датчик конвейера 2",   // "FB_DI"
                           "On/Off_Filters_DI" := "DI".DI_9."bFiltr_on/off",
                           Set_Time_Dely := "DI".DI_9.diTime_filtr,
                           Simulate := "DI".DI_9.bSimulation,
                           Simulate_Value := "DI".DI_9."bSim_On/Off",
                           Value => "Alarms".xSensorConveyorZator_2);
END_REGION

REGION Network 11: Работа чатотника - 1
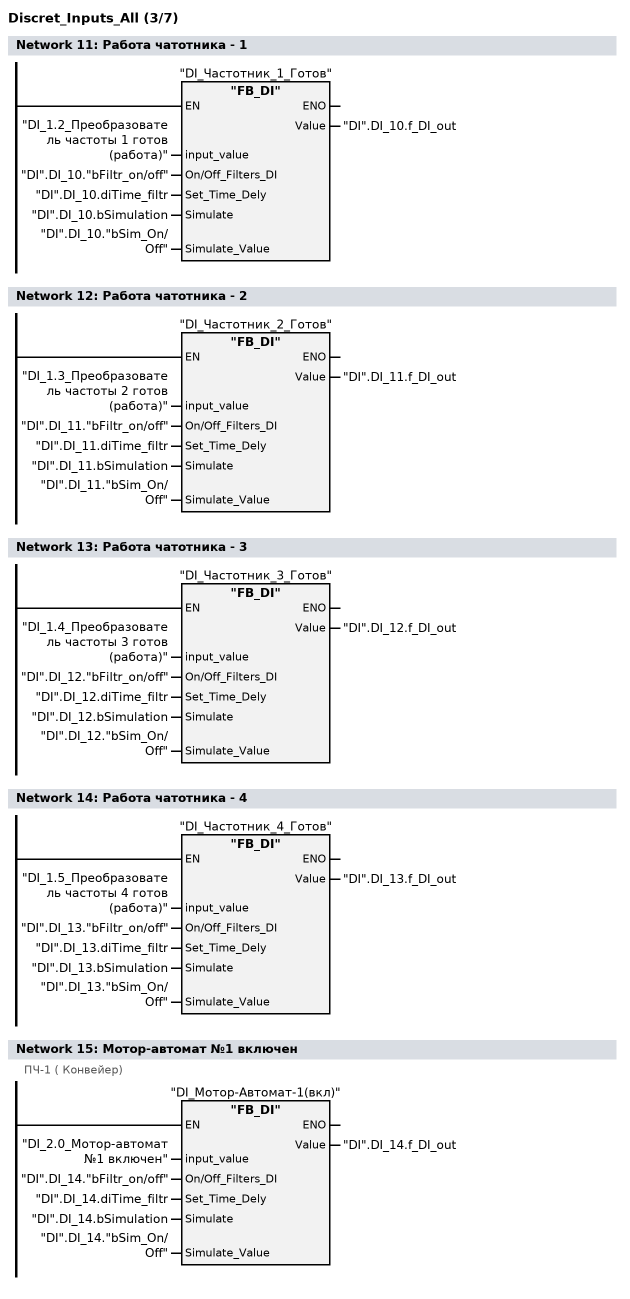
   RUNG wire#powerrail
      "DI_Частотник_1_Готов"(input_value := "DI_1.2_Преобразователь частоты 1 готов (работа)", "On/Off_Filters_DI" := "DI".DI_10."bFiltr_on/off", Set_Time_Dely := "DI".DI_10.diTime_filtr, Simulate := "DI".DI_10.bSimulation, Simulate_Value := "DI".DI_10."bSim_On/Off", Value => "DI".DI_10.f_DI_out)
   END_RUNG
   // the same network as SCL:
   "DI_Частотник_1_Готов"(input_value := "DI_1.2_Преобразователь частоты 1 готов (работа)",   // "FB_DI"
                          "On/Off_Filters_DI" := "DI".DI_10."bFiltr_on/off",
                          Set_Time_Dely := "DI".DI_10.diTime_filtr,
                          Simulate := "DI".DI_10.bSimulation,
                          Simulate_Value := "DI".DI_10."bSim_On/Off",
                          Value => "DI".DI_10.f_DI_out);
END_REGION

REGION Network 12: Работа чатотника - 2
   RUNG wire#powerrail
      "DI_Частотник_2_Готов"(input_value := "DI_1.3_Преобразователь частоты 2 готов (работа)", "On/Off_Filters_DI" := "DI".DI_11."bFiltr_on/off", Set_Time_Dely := "DI".DI_11.diTime_filtr, Simulate := "DI".DI_11.bSimulation, Simulate_Value := "DI".DI_11."bSim_On/Off", Value => "DI".DI_11.f_DI_out)
   END_RUNG
   // the same network as SCL:
   "DI_Частотник_2_Готов"(input_value := "DI_1.3_Преобразователь частоты 2 готов (работа)",   // "FB_DI"
                          "On/Off_Filters_DI" := "DI".DI_11."bFiltr_on/off",
                          Set_Time_Dely := "DI".DI_11.diTime_filtr,
                          Simulate := "DI".DI_11.bSimulation,
                          Simulate_Value := "DI".DI_11."bSim_On/Off",
                          Value => "DI".DI_11.f_DI_out);
END_REGION

REGION Network 13: Работа чатотника - 3
   RUNG wire#powerrail
      "DI_Частотник_3_Готов"(input_value := "DI_1.4_Преобразователь частоты 3 готов (работа)", "On/Off_Filters_DI" := "DI".DI_12."bFiltr_on/off", Set_Time_Dely := "DI".DI_12.diTime_filtr, Simulate := "DI".DI_12.bSimulation, Simulate_Value := "DI".DI_12."bSim_On/Off", Value => "DI".DI_12.f_DI_out)
   END_RUNG
   // the same network as SCL:
   "DI_Частотник_3_Готов"(input_value := "DI_1.4_Преобразователь частоты 3 готов (работа)",   // "FB_DI"
                          "On/Off_Filters_DI" := "DI".DI_12."bFiltr_on/off",
                          Set_Time_Dely := "DI".DI_12.diTime_filtr,
                          Simulate := "DI".DI_12.bSimulation,
                          Simulate_Value := "DI".DI_12."bSim_On/Off",
                          Value => "DI".DI_12.f_DI_out);
END_REGION

REGION Network 14: Работа чатотника - 4
   RUNG wire#powerrail
      "DI_Частотник_4_Готов"(input_value := "DI_1.5_Преобразователь частоты 4 готов (работа)", "On/Off_Filters_DI" := "DI".DI_13."bFiltr_on/off", Set_Time_Dely := "DI".DI_13.diTime_filtr, Simulate := "DI".DI_13.bSimulation, Simulate_Value := "DI".DI_13."bSim_On/Off", Value => "DI".DI_13.f_DI_out)
   END_RUNG
   // the same network as SCL:
   "DI_Частотник_4_Готов"(input_value := "DI_1.5_Преобразователь частоты 4 готов (работа)",   // "FB_DI"
                          "On/Off_Filters_DI" := "DI".DI_13."bFiltr_on/off",
                          Set_Time_Dely := "DI".DI_13.diTime_filtr,
                          Simulate := "DI".DI_13.bSimulation,
                          Simulate_Value := "DI".DI_13."bSim_On/Off",
                          Value => "DI".DI_13.f_DI_out);
END_REGION

REGION Network 15: Мотор-автомат №1 включен
   // ПЧ-1 ( Конвейер)
   RUNG wire#powerrail
      "DI_Мотор-Автомат-1(вкл)"(input_value := "DI_2.0_Мотор-автомат №1 включен", "On/Off_Filters_DI" := "DI".DI_14."bFiltr_on/off", Set_Time_Dely := "DI".DI_14.diTime_filtr, Simulate := "DI".DI_14.bSimulation, Simulate_Value := "DI".DI_14."bSim_On/Off", Value => "DI".DI_14.f_DI_out)
   END_RUNG
   // the same network as SCL:
   "DI_Мотор-Автомат-1(вкл)"(input_value := "DI_2.0_Мотор-автомат №1 включен",   // "FB_DI"
                           "On/Off_Filters_DI" := "DI".DI_14."bFiltr_on/off",
                           Set_Time_Dely := "DI".DI_14.diTime_filtr,
                           Simulate := "DI".DI_14.bSimulation,
                           Simulate_Value := "DI".DI_14."bSim_On/Off",
                           Value => "DI".DI_14.f_DI_out);
END_REGION

REGION Network 16: Мотор-автомат №2 включен
   // ПЧ-2 ( Конвейер)
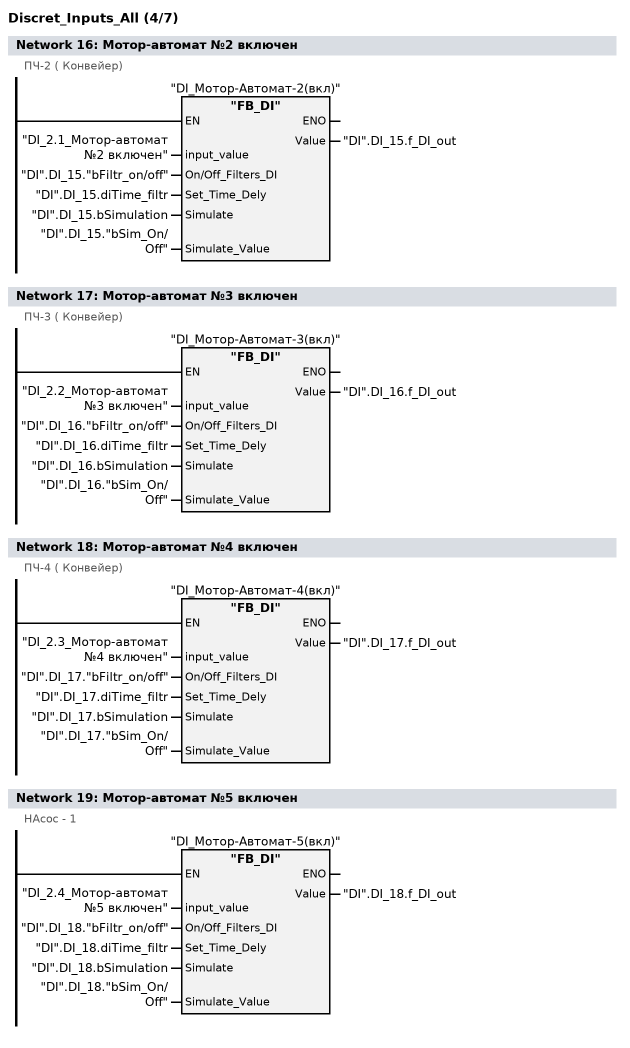
   RUNG wire#powerrail
      "DI_Мотор-Автомат-2(вкл)"(input_value := "DI_2.1_Мотор-автомат №2 включен", "On/Off_Filters_DI" := "DI".DI_15."bFiltr_on/off", Set_Time_Dely := "DI".DI_15.diTime_filtr, Simulate := "DI".DI_15.bSimulation, Simulate_Value := "DI".DI_15."bSim_On/Off", Value => "DI".DI_15.f_DI_out)
   END_RUNG
   // the same network as SCL:
   "DI_Мотор-Автомат-2(вкл)"(input_value := "DI_2.1_Мотор-автомат №2 включен",   // "FB_DI"
                           "On/Off_Filters_DI" := "DI".DI_15."bFiltr_on/off",
                           Set_Time_Dely := "DI".DI_15.diTime_filtr,
                           Simulate := "DI".DI_15.bSimulation,
                           Simulate_Value := "DI".DI_15."bSim_On/Off",
                           Value => "DI".DI_15.f_DI_out);
END_REGION

REGION Network 17: Мотор-автомат №3 включен
   // ПЧ-3 ( Конвейер)
   RUNG wire#powerrail
      "DI_Мотор-Автомат-3(вкл)"(input_value := "DI_2.2_Мотор-автомат №3 включен", "On/Off_Filters_DI" := "DI".DI_16."bFiltr_on/off", Set_Time_Dely := "DI".DI_16.diTime_filtr, Simulate := "DI".DI_16.bSimulation, Simulate_Value := "DI".DI_16."bSim_On/Off", Value => "DI".DI_16.f_DI_out)
   END_RUNG
   // the same network as SCL:
   "DI_Мотор-Автомат-3(вкл)"(input_value := "DI_2.2_Мотор-автомат №3 включен",   // "FB_DI"
                           "On/Off_Filters_DI" := "DI".DI_16."bFiltr_on/off",
                           Set_Time_Dely := "DI".DI_16.diTime_filtr,
                           Simulate := "DI".DI_16.bSimulation,
                           Simulate_Value := "DI".DI_16."bSim_On/Off",
                           Value => "DI".DI_16.f_DI_out);
END_REGION

REGION Network 18: Мотор-автомат №4 включен
   // ПЧ-4 ( Конвейер)
   RUNG wire#powerrail
      "DI_Мотор-Автомат-4(вкл)"(input_value := "DI_2.3_Мотор-автомат №4 включен", "On/Off_Filters_DI" := "DI".DI_17."bFiltr_on/off", Set_Time_Dely := "DI".DI_17.diTime_filtr, Simulate := "DI".DI_17.bSimulation, Simulate_Value := "DI".DI_17."bSim_On/Off", Value => "DI".DI_17.f_DI_out)
   END_RUNG
   // the same network as SCL:
   "DI_Мотор-Автомат-4(вкл)"(input_value := "DI_2.3_Мотор-автомат №4 включен",   // "FB_DI"
                           "On/Off_Filters_DI" := "DI".DI_17."bFiltr_on/off",
                           Set_Time_Dely := "DI".DI_17.diTime_filtr,
                           Simulate := "DI".DI_17.bSimulation,
                           Simulate_Value := "DI".DI_17."bSim_On/Off",
                           Value => "DI".DI_17.f_DI_out);
END_REGION

REGION Network 19: Мотор-автомат №5 включен
   // НАсос - 1
   RUNG wire#powerrail
      "DI_Мотор-Автомат-5(вкл)"(input_value := "DI_2.4_Мотор-автомат №5 включен", "On/Off_Filters_DI" := "DI".DI_18."bFiltr_on/off", Set_Time_Dely := "DI".DI_18.diTime_filtr, Simulate := "DI".DI_18.bSimulation, Simulate_Value := "DI".DI_18."bSim_On/Off", Value => "DI".DI_18.f_DI_out)
   END_RUNG
   // the same network as SCL:
   "DI_Мотор-Автомат-5(вкл)"(input_value := "DI_2.4_Мотор-автомат №5 включен",   // "FB_DI"
                           "On/Off_Filters_DI" := "DI".DI_18."bFiltr_on/off",
                           Set_Time_Dely := "DI".DI_18.diTime_filtr,
                           Simulate := "DI".DI_18.bSimulation,
                           Simulate_Value := "DI".DI_18."bSim_On/Off",
                           Value => "DI".DI_18.f_DI_out);
END_REGION

REGION Network 20: Мотор-автомат №6 включен
   // НАсос - 2
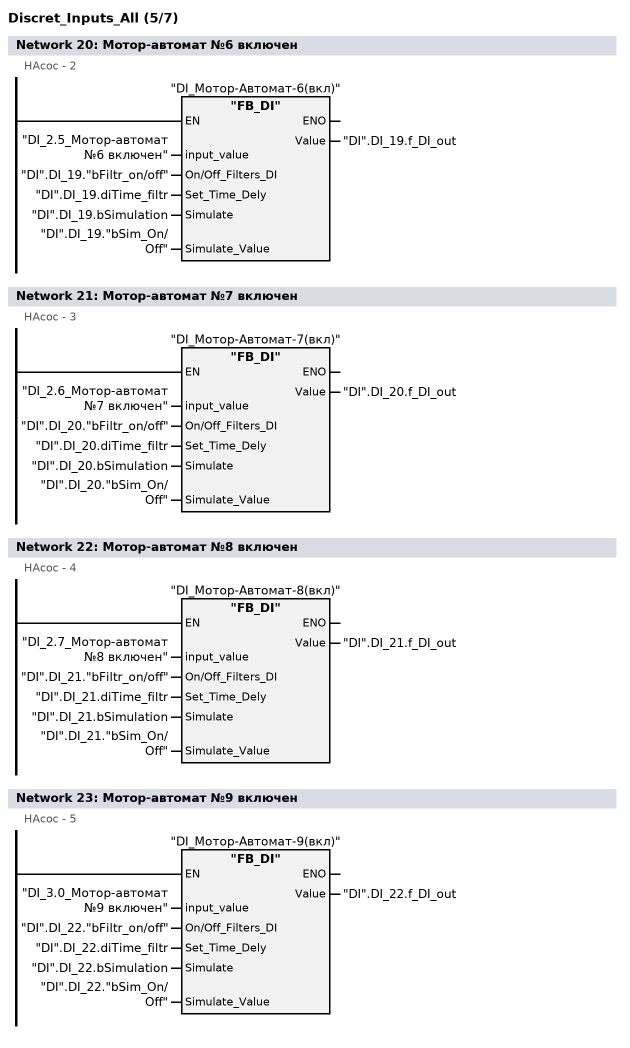
   RUNG wire#powerrail
      "DI_Мотор-Автомат-6(вкл)"(input_value := "DI_2.5_Мотор-автомат №6 включен", "On/Off_Filters_DI" := "DI".DI_19."bFiltr_on/off", Set_Time_Dely := "DI".DI_19.diTime_filtr, Simulate := "DI".DI_19.bSimulation, Simulate_Value := "DI".DI_19."bSim_On/Off", Value => "DI".DI_19.f_DI_out)
   END_RUNG
   // the same network as SCL:
   "DI_Мотор-Автомат-6(вкл)"(input_value := "DI_2.5_Мотор-автомат №6 включен",   // "FB_DI"
                           "On/Off_Filters_DI" := "DI".DI_19."bFiltr_on/off",
                           Set_Time_Dely := "DI".DI_19.diTime_filtr,
                           Simulate := "DI".DI_19.bSimulation,
                           Simulate_Value := "DI".DI_19."bSim_On/Off",
                           Value => "DI".DI_19.f_DI_out);
END_REGION

REGION Network 21: Мотор-автомат №7 включен
   // НАсос - 3
   RUNG wire#powerrail
      "DI_Мотор-Автомат-7(вкл)"(input_value := "DI_2.6_Мотор-автомат №7 включен", "On/Off_Filters_DI" := "DI".DI_20."bFiltr_on/off", Set_Time_Dely := "DI".DI_20.diTime_filtr, Simulate := "DI".DI_20.bSimulation, Simulate_Value := "DI".DI_20."bSim_On/Off", Value => "DI".DI_20.f_DI_out)
   END_RUNG
   // the same network as SCL:
   "DI_Мотор-Автомат-7(вкл)"(input_value := "DI_2.6_Мотор-автомат №7 включен",   // "FB_DI"
                           "On/Off_Filters_DI" := "DI".DI_20."bFiltr_on/off",
                           Set_Time_Dely := "DI".DI_20.diTime_filtr,
                           Simulate := "DI".DI_20.bSimulation,
                           Simulate_Value := "DI".DI_20."bSim_On/Off",
                           Value => "DI".DI_20.f_DI_out);
END_REGION

REGION Network 22: Мотор-автомат №8 включен
   // НАсос - 4
   RUNG wire#powerrail
      "DI_Мотор-Автомат-8(вкл)"(input_value := "DI_2.7_Мотор-автомат №8 включен", "On/Off_Filters_DI" := "DI".DI_21."bFiltr_on/off", Set_Time_Dely := "DI".DI_21.diTime_filtr, Simulate := "DI".DI_21.bSimulation, Simulate_Value := "DI".DI_21."bSim_On/Off", Value => "DI".DI_21.f_DI_out)
   END_RUNG
   // the same network as SCL:
   "DI_Мотор-Автомат-8(вкл)"(input_value := "DI_2.7_Мотор-автомат №8 включен",   // "FB_DI"
                           "On/Off_Filters_DI" := "DI".DI_21."bFiltr_on/off",
                           Set_Time_Dely := "DI".DI_21.diTime_filtr,
                           Simulate := "DI".DI_21.bSimulation,
                           Simulate_Value := "DI".DI_21."bSim_On/Off",
                           Value => "DI".DI_21.f_DI_out);
END_REGION

REGION Network 23: Мотор-автомат №9 включен
   // НАсос - 5
   RUNG wire#powerrail
      "DI_Мотор-Автомат-9(вкл)"(input_value := "DI_3.0_Мотор-автомат №9 включен", "On/Off_Filters_DI" := "DI".DI_22."bFiltr_on/off", Set_Time_Dely := "DI".DI_22.diTime_filtr, Simulate := "DI".DI_22.bSimulation, Simulate_Value := "DI".DI_22."bSim_On/Off", Value => "DI".DI_22.f_DI_out)
   END_RUNG
   // the same network as SCL:
   "DI_Мотор-Автомат-9(вкл)"(input_value := "DI_3.0_Мотор-автомат №9 включен",   // "FB_DI"
                           "On/Off_Filters_DI" := "DI".DI_22."bFiltr_on/off",
                           Set_Time_Dely := "DI".DI_22.diTime_filtr,
                           Simulate := "DI".DI_22.bSimulation,
                           Simulate_Value := "DI".DI_22."bSim_On/Off",
                           Value => "DI".DI_22.f_DI_out);
END_REGION

REGION Network 24: Мотор-автомат №10 включен
   // Воздух - ветродуйка
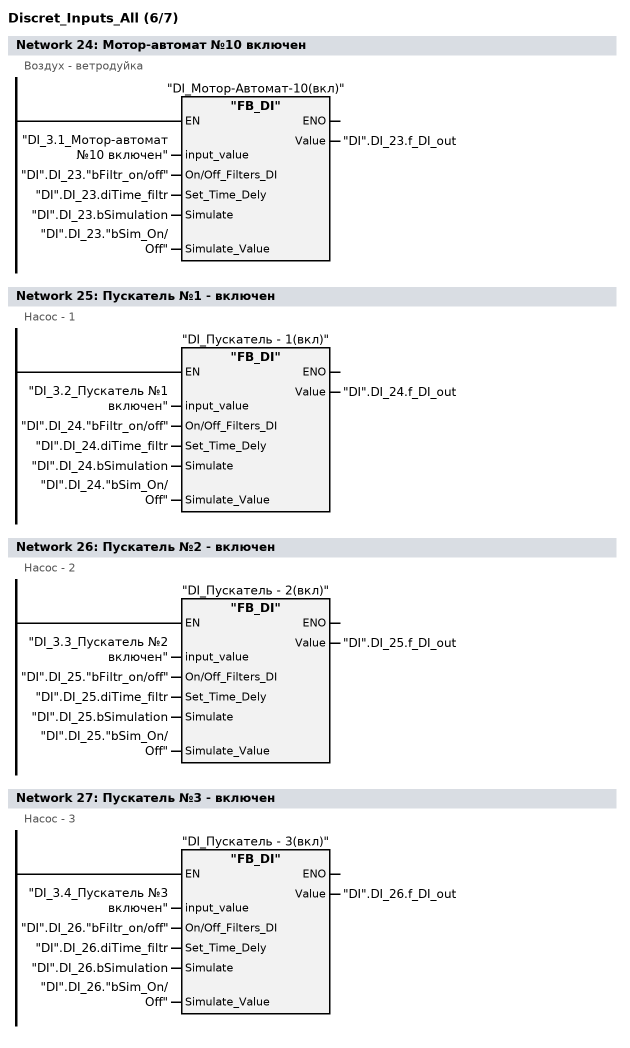
   RUNG wire#powerrail
      "DI_Мотор-Автомат-10(вкл)"(input_value := "DI_3.1_Мотор-автомат №10 включен", "On/Off_Filters_DI" := "DI".DI_23."bFiltr_on/off", Set_Time_Dely := "DI".DI_23.diTime_filtr, Simulate := "DI".DI_23.bSimulation, Simulate_Value := "DI".DI_23."bSim_On/Off", Value => "DI".DI_23.f_DI_out)
   END_RUNG
   // the same network as SCL:
   "DI_Мотор-Автомат-10(вкл)"(input_value := "DI_3.1_Мотор-автомат №10 включен",   // "FB_DI"
                           "On/Off_Filters_DI" := "DI".DI_23."bFiltr_on/off",
                           Set_Time_Dely := "DI".DI_23.diTime_filtr,
                           Simulate := "DI".DI_23.bSimulation,
                           Simulate_Value := "DI".DI_23."bSim_On/Off",
                           Value => "DI".DI_23.f_DI_out);
END_REGION

REGION Network 25: Пускатель №1 - включен
   // Насос - 1
   RUNG wire#powerrail
      "DI_Пускатель - 1(вкл)"(input_value := "DI_3.2_Пускатель №1 включен", "On/Off_Filters_DI" := "DI".DI_24."bFiltr_on/off", Set_Time_Dely := "DI".DI_24.diTime_filtr, Simulate := "DI".DI_24.bSimulation, Simulate_Value := "DI".DI_24."bSim_On/Off", Value => "DI".DI_24.f_DI_out)
   END_RUNG
   // the same network as SCL:
   "DI_Пускатель - 1(вкл)"(input_value := "DI_3.2_Пускатель №1 включен",   // "FB_DI"
                           "On/Off_Filters_DI" := "DI".DI_24."bFiltr_on/off",
                           Set_Time_Dely := "DI".DI_24.diTime_filtr,
                           Simulate := "DI".DI_24.bSimulation,
                           Simulate_Value := "DI".DI_24."bSim_On/Off",
                           Value => "DI".DI_24.f_DI_out);
END_REGION

REGION Network 26: Пускатель №2 - включен
   // Насос - 2
   RUNG wire#powerrail
      "DI_Пускатель - 2(вкл)"(input_value := "DI_3.3_Пускатель №2 включен", "On/Off_Filters_DI" := "DI".DI_25."bFiltr_on/off", Set_Time_Dely := "DI".DI_25.diTime_filtr, Simulate := "DI".DI_25.bSimulation, Simulate_Value := "DI".DI_25."bSim_On/Off", Value => "DI".DI_25.f_DI_out)
   END_RUNG
   // the same network as SCL:
   "DI_Пускатель - 2(вкл)"(input_value := "DI_3.3_Пускатель №2 включен",   // "FB_DI"
                           "On/Off_Filters_DI" := "DI".DI_25."bFiltr_on/off",
                           Set_Time_Dely := "DI".DI_25.diTime_filtr,
                           Simulate := "DI".DI_25.bSimulation,
                           Simulate_Value := "DI".DI_25."bSim_On/Off",
                           Value => "DI".DI_25.f_DI_out);
END_REGION

REGION Network 27: Пускатель №3 - включен
   // Насос - 3
   RUNG wire#powerrail
      "DI_Пускатель - 3(вкл)"(input_value := "DI_3.4_Пускатель №3 включен", "On/Off_Filters_DI" := "DI".DI_26."bFiltr_on/off", Set_Time_Dely := "DI".DI_26.diTime_filtr, Simulate := "DI".DI_26.bSimulation, Simulate_Value := "DI".DI_26."bSim_On/Off", Value => "DI".DI_26.f_DI_out)
   END_RUNG
   // the same network as SCL:
   "DI_Пускатель - 3(вкл)"(input_value := "DI_3.4_Пускатель №3 включен",   // "FB_DI"
                           "On/Off_Filters_DI" := "DI".DI_26."bFiltr_on/off",
                           Set_Time_Dely := "DI".DI_26.diTime_filtr,
                           Simulate := "DI".DI_26.bSimulation,
                           Simulate_Value := "DI".DI_26."bSim_On/Off",
                           Value => "DI".DI_26.f_DI_out);
END_REGION

REGION Network 28: Пускатель №4 - включен
   // Насос - 4
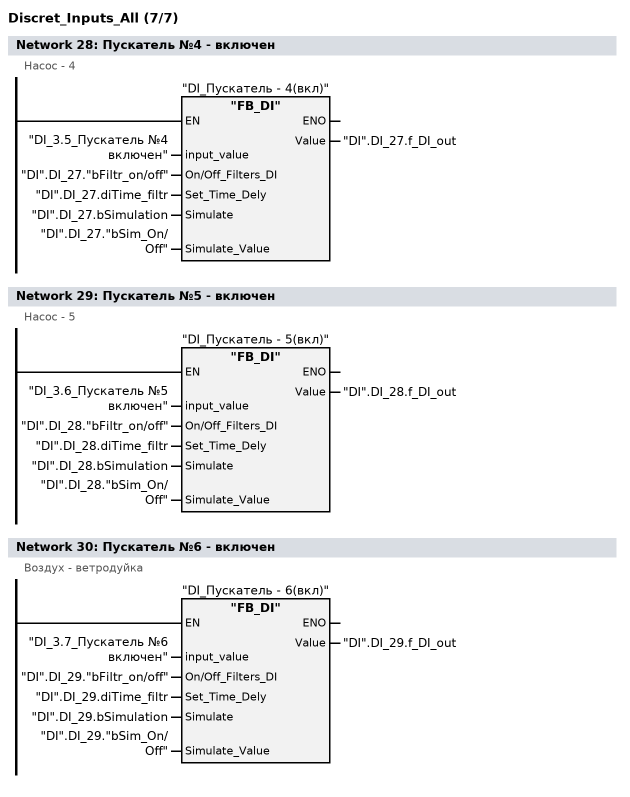
   RUNG wire#powerrail
      "DI_Пускатель - 4(вкл)"(input_value := "DI_3.5_Пускатель №4 включен", "On/Off_Filters_DI" := "DI".DI_27."bFiltr_on/off", Set_Time_Dely := "DI".DI_27.diTime_filtr, Simulate := "DI".DI_27.bSimulation, Simulate_Value := "DI".DI_27."bSim_On/Off", Value => "DI".DI_27.f_DI_out)
   END_RUNG
   // the same network as SCL:
   "DI_Пускатель - 4(вкл)"(input_value := "DI_3.5_Пускатель №4 включен",   // "FB_DI"
                           "On/Off_Filters_DI" := "DI".DI_27."bFiltr_on/off",
                           Set_Time_Dely := "DI".DI_27.diTime_filtr,
                           Simulate := "DI".DI_27.bSimulation,
                           Simulate_Value := "DI".DI_27."bSim_On/Off",
                           Value => "DI".DI_27.f_DI_out);
END_REGION

REGION Network 29: Пускатель №5 - включен
   // Насос - 5
   RUNG wire#powerrail
      "DI_Пускатель - 5(вкл)"(input_value := "DI_3.6_Пускатель №5 включен", "On/Off_Filters_DI" := "DI".DI_28."bFiltr_on/off", Set_Time_Dely := "DI".DI_28.diTime_filtr, Simulate := "DI".DI_28.bSimulation, Simulate_Value := "DI".DI_28."bSim_On/Off", Value => "DI".DI_28.f_DI_out)
   END_RUNG
   // the same network as SCL:
   "DI_Пускатель - 5(вкл)"(input_value := "DI_3.6_Пускатель №5 включен",   // "FB_DI"
                           "On/Off_Filters_DI" := "DI".DI_28."bFiltr_on/off",
                           Set_Time_Dely := "DI".DI_28.diTime_filtr,
                           Simulate := "DI".DI_28.bSimulation,
                           Simulate_Value := "DI".DI_28."bSim_On/Off",
                           Value => "DI".DI_28.f_DI_out);
END_REGION

REGION Network 30: Пускатель №6 - включен
   // Воздух - ветродуйка
   RUNG wire#powerrail
      "DI_Пускатель - 6(вкл)"(input_value := "DI_3.7_Пускатель №6 включен", "On/Off_Filters_DI" := "DI".DI_29."bFiltr_on/off", Set_Time_Dely := "DI".DI_29.diTime_filtr, Simulate := "DI".DI_29.bSimulation, Simulate_Value := "DI".DI_29."bSim_On/Off", Value => "DI".DI_29.f_DI_out)
   END_RUNG
   // the same network as SCL:
   "DI_Пускатель - 6(вкл)"(input_value := "DI_3.7_Пускатель №6 включен",   // "FB_DI"
                           "On/Off_Filters_DI" := "DI".DI_29."bFiltr_on/off",
                           Set_Time_Dely := "DI".DI_29.diTime_filtr,
                           Simulate := "DI".DI_29.bSimulation,
                           Simulate_Value := "DI".DI_29."bSim_On/Off",
                           Value => "DI".DI_29.f_DI_out);
END_REGION
END_FUNCTION

FUNCTION "Конвейера" : Void   // FC9, LAD
{ S7_Optimized_Access := 'TRUE' }
VERSION : 0.1
// Блоки для управления "Конвейерами"
BEGIN

REGION Network 1: Конвейер - 1
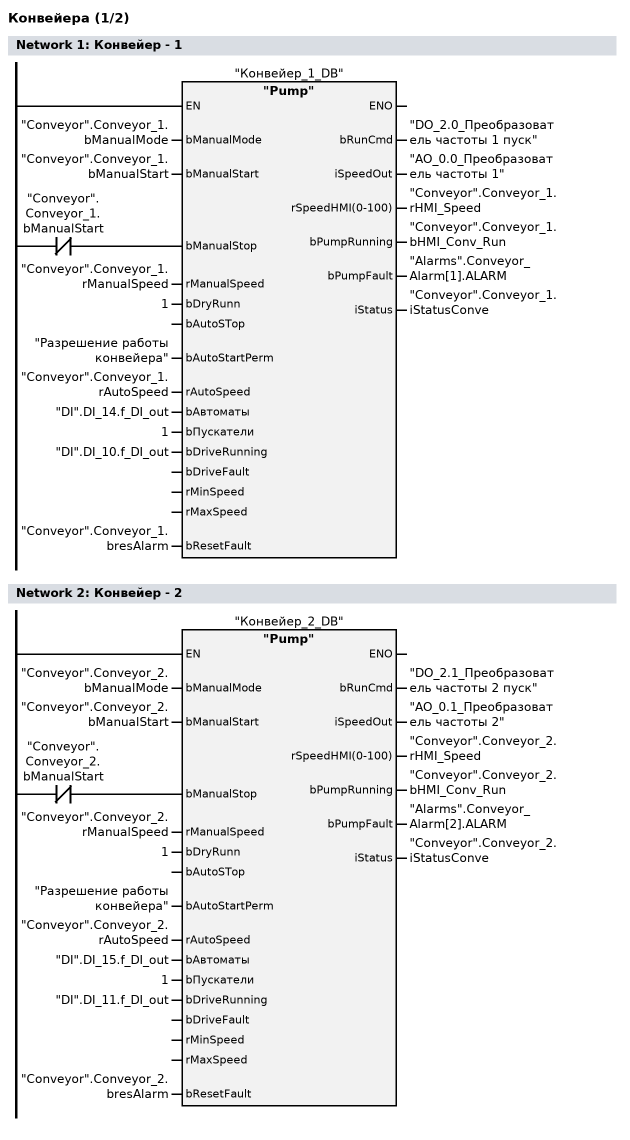
   RUNG wire#powerrail
      "Конвейер_1_DB"(bManualStop := wire#w1, bManualMode := "Conveyor".Conveyor_1.bManualMode, bManualStart := "Conveyor".Conveyor_1.bManualStart, rManualSpeed := "Conveyor".Conveyor_1.rManualSpeed, bDryRunn := 1, bAutoStartPerm := "Разрешение работы конвейера", rAutoSpeed := "Conveyor".Conveyor_1.rAutoSpeed, bАвтоматы := "DI".DI_14.f_DI_out, bПускатели := 1, bDriveRunning := "DI".DI_10.f_DI_out, bDriveFault :=, rMinSpeed :=, rMaxSpeed :=, bResetFault := "Conveyor".Conveyor_1.bresAlarm, bRunCmd => "DO_2.0_Преобразователь частоты 1 пуск", iSpeedOut => "AO_0.0_Преобразователь частоты 1", "rSpeedHMI(0-100)" => "Conveyor".Conveyor_1.rHMI_Speed, bPumpRunning => "Conveyor".Conveyor_1.bHMI_Conv_Run, bPumpFault => "Alarms".Conveyor_Alarm[1].ALARM, iStatus => "Conveyor".Conveyor_1.iStatusConve, bAutoSTop :=)
   END_RUNG
   RUNG wire#powerrail
      I_Contact( "Conveyor".Conveyor_1.bManualStart )
   END_RUNG wire#w1
   // the same network as SCL:
   "Конвейер_1_DB"(bManualMode := "Conveyor".Conveyor_1.bManualMode,   // "Pump"
                   bManualStart := "Conveyor".Conveyor_1.bManualStart,
                   bManualStop := NOT "Conveyor".Conveyor_1.bManualStart,
                   rManualSpeed := "Conveyor".Conveyor_1.rManualSpeed,
                   bDryRunn := 1,
                   bAutoStartPerm := "Разрешение работы конвейера",
                   rAutoSpeed := "Conveyor".Conveyor_1.rAutoSpeed,
                   bАвтоматы := "DI".DI_14.f_DI_out,
                   bПускатели := 1,
                   bDriveRunning := "DI".DI_10.f_DI_out,
                   bResetFault := "Conveyor".Conveyor_1.bresAlarm,
                   bRunCmd => "DO_2.0_Преобразователь частоты 1 пуск",
                   iSpeedOut => "AO_0.0_Преобразователь частоты 1",
                   "rSpeedHMI(0-100)" => "Conveyor".Conveyor_1.rHMI_Speed,
                   bPumpRunning => "Conveyor".Conveyor_1.bHMI_Conv_Run,
                   bPumpFault => "Alarms".Conveyor_Alarm[1].ALARM,
                   iStatus => "Conveyor".Conveyor_1.iStatusConve);
END_REGION

REGION Network 2: Конвейер - 2
   RUNG wire#powerrail
      "Конвейер_2_DB"(bManualStop := wire#w1, bManualMode := "Conveyor".Conveyor_2.bManualMode, bManualStart := "Conveyor".Conveyor_2.bManualStart, rManualSpeed := "Conveyor".Conveyor_2.rManualSpeed, bDryRunn := 1, bAutoStartPerm := "Разрешение работы конвейера", rAutoSpeed := "Conveyor".Conveyor_2.rAutoSpeed, bАвтоматы := "DI".DI_15.f_DI_out, bПускатели := 1, bDriveRunning := "DI".DI_11.f_DI_out, bDriveFault :=, rMinSpeed :=, rMaxSpeed :=, bResetFault := "Conveyor".Conveyor_2.bresAlarm, bRunCmd => "DO_2.1_Преобразователь частоты 2 пуск", iSpeedOut => "AO_0.1_Преобразователь частоты 2", "rSpeedHMI(0-100)" => "Conveyor".Conveyor_2.rHMI_Speed, bPumpRunning => "Conveyor".Conveyor_2.bHMI_Conv_Run, bPumpFault => "Alarms".Conveyor_Alarm[2].ALARM, iStatus => "Conveyor".Conveyor_2.iStatusConve, bAutoSTop :=)
   END_RUNG
   RUNG wire#powerrail
      I_Contact( "Conveyor".Conveyor_2.bManualStart )
   END_RUNG wire#w1
   // the same network as SCL:
   "Конвейер_2_DB"(bManualMode := "Conveyor".Conveyor_2.bManualMode,   // "Pump"
                   bManualStart := "Conveyor".Conveyor_2.bManualStart,
                   bManualStop := NOT "Conveyor".Conveyor_2.bManualStart,
                   rManualSpeed := "Conveyor".Conveyor_2.rManualSpeed,
                   bDryRunn := 1,
                   bAutoStartPerm := "Разрешение работы конвейера",
                   rAutoSpeed := "Conveyor".Conveyor_2.rAutoSpeed,
                   bАвтоматы := "DI".DI_15.f_DI_out,
                   bПускатели := 1,
                   bDriveRunning := "DI".DI_11.f_DI_out,
                   bResetFault := "Conveyor".Conveyor_2.bresAlarm,
                   bRunCmd => "DO_2.1_Преобразователь частоты 2 пуск",
                   iSpeedOut => "AO_0.1_Преобразователь частоты 2",
                   "rSpeedHMI(0-100)" => "Conveyor".Conveyor_2.rHMI_Speed,
                   bPumpRunning => "Conveyor".Conveyor_2.bHMI_Conv_Run,
                   bPumpFault => "Alarms".Conveyor_Alarm[2].ALARM,
                   iStatus => "Conveyor".Conveyor_2.iStatusConve);
END_REGION

REGION Network 3: Конвейер - 3
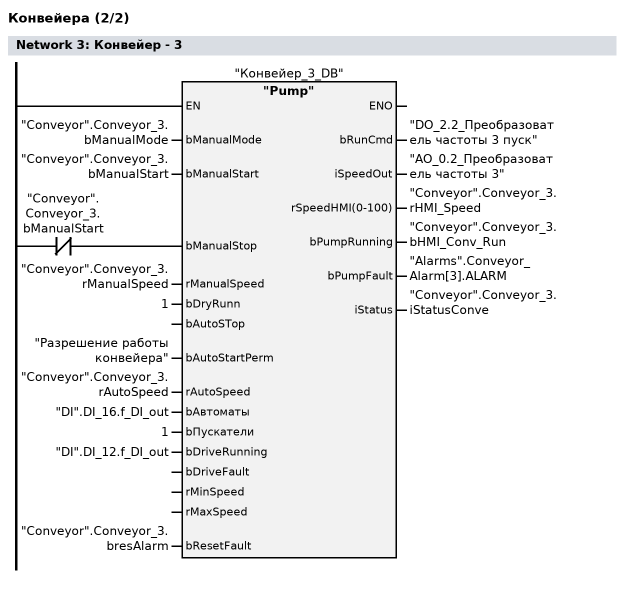
   RUNG wire#powerrail
      "Конвейер_3_DB"(bManualStop := wire#w1, bManualMode := "Conveyor".Conveyor_3.bManualMode, bManualStart := "Conveyor".Conveyor_3.bManualStart, rManualSpeed := "Conveyor".Conveyor_3.rManualSpeed, bDryRunn := 1, bAutoStartPerm := "Разрешение работы конвейера", rAutoSpeed := "Conveyor".Conveyor_3.rAutoSpeed, bАвтоматы := "DI".DI_16.f_DI_out, bПускатели := 1, bDriveRunning := "DI".DI_12.f_DI_out, bDriveFault :=, rMinSpeed :=, rMaxSpeed :=, bResetFault := "Conveyor".Conveyor_3.bresAlarm, bRunCmd => "DO_2.2_Преобразователь частоты 3 пуск", iSpeedOut => "AO_0.2_Преобразователь частоты 3", "rSpeedHMI(0-100)" => "Conveyor".Conveyor_3.rHMI_Speed, bPumpRunning => "Conveyor".Conveyor_3.bHMI_Conv_Run, bPumpFault => "Alarms".Conveyor_Alarm[3].ALARM, iStatus => "Conveyor".Conveyor_3.iStatusConve, bAutoSTop :=)
   END_RUNG
   RUNG wire#powerrail
      I_Contact( "Conveyor".Conveyor_3.bManualStart )
   END_RUNG wire#w1
   // the same network as SCL:
   "Конвейер_3_DB"(bManualMode := "Conveyor".Conveyor_3.bManualMode,   // "Pump"
                   bManualStart := "Conveyor".Conveyor_3.bManualStart,
                   bManualStop := NOT "Conveyor".Conveyor_3.bManualStart,
                   rManualSpeed := "Conveyor".Conveyor_3.rManualSpeed,
                   bDryRunn := 1,
                   bAutoStartPerm := "Разрешение работы конвейера",
                   rAutoSpeed := "Conveyor".Conveyor_3.rAutoSpeed,
                   bАвтоматы := "DI".DI_16.f_DI_out,
                   bПускатели := 1,
                   bDriveRunning := "DI".DI_12.f_DI_out,
                   bResetFault := "Conveyor".Conveyor_3.bresAlarm,
                   bRunCmd => "DO_2.2_Преобразователь частоты 3 пуск",
                   iSpeedOut => "AO_0.2_Преобразователь частоты 3",
                   "rSpeedHMI(0-100)" => "Conveyor".Conveyor_3.rHMI_Speed,
                   bPumpRunning => "Conveyor".Conveyor_3.bHMI_Conv_Run,
                   bPumpFault => "Alarms".Conveyor_Alarm[3].ALARM,
                   iStatus => "Conveyor".Conveyor_3.iStatusConve);
END_REGION
END_FUNCTION

FUNCTION "Вентилятор" : Void   // FC10, LAD
{ S7_Optimized_Access := 'TRUE' }
VERSION : 0.1
// Управление вентилятором
BEGIN

REGION Network 1: Вентилятор
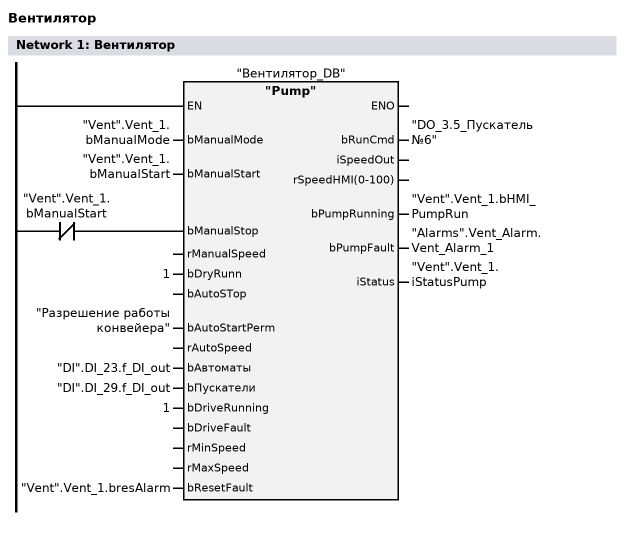
   RUNG wire#powerrail
      "Вентилятор_DB"(bManualStop := wire#w1, bManualMode := "Vent".Vent_1.bManualMode, bManualStart := "Vent".Vent_1.bManualStart, rManualSpeed :=, bDryRunn := 1, bAutoStartPerm := "Разрешение работы конвейера", rAutoSpeed :=, bАвтоматы := "DI".DI_23.f_DI_out, bПускатели := "DI".DI_29.f_DI_out, bDriveRunning := 1, bDriveFault :=, rMinSpeed :=, rMaxSpeed :=, bResetFault := "Vent".Vent_1.bresAlarm, bRunCmd => "DO_3.5_Пускатель №6", iSpeedOut =>, "rSpeedHMI(0-100)" =>, bPumpRunning => "Vent".Vent_1.bHMI_PumpRun, bPumpFault => "Alarms".Vent_Alarm.Vent_Alarm_1, iStatus => "Vent".Vent_1.iStatusPump, bAutoSTop :=)
   END_RUNG
   RUNG wire#powerrail
      I_Contact( "Vent".Vent_1.bManualStart )
   END_RUNG wire#w1
   // the same network as SCL:
   "Вентилятор_DB"(bManualMode := "Vent".Vent_1.bManualMode,   // "Pump"
                   bManualStart := "Vent".Vent_1.bManualStart,
                   bManualStop := NOT "Vent".Vent_1.bManualStart,
                   bDryRunn := 1,
                   bAutoStartPerm := "Разрешение работы конвейера",
                   bАвтоматы := "DI".DI_23.f_DI_out,
                   bПускатели := "DI".DI_29.f_DI_out,
                   bDriveRunning := 1,
                   bResetFault := "Vent".Vent_1.bresAlarm,
                   bRunCmd => "DO_3.5_Пускатель №6",
                   bPumpRunning => "Vent".Vent_1.bHMI_PumpRun,
                   bPumpFault => "Alarms".Vent_Alarm.Vent_Alarm_1,
                   iStatus => "Vent".Vent_1.iStatusPump);
END_REGION
END_FUNCTION

FUNCTION "Наполнение емкостей" : Void   // FC11, LAD
{ S7_Optimized_Access := 'TRUE' }
VERSION : 0.1
BEGIN

REGION Network 1: Бак 1
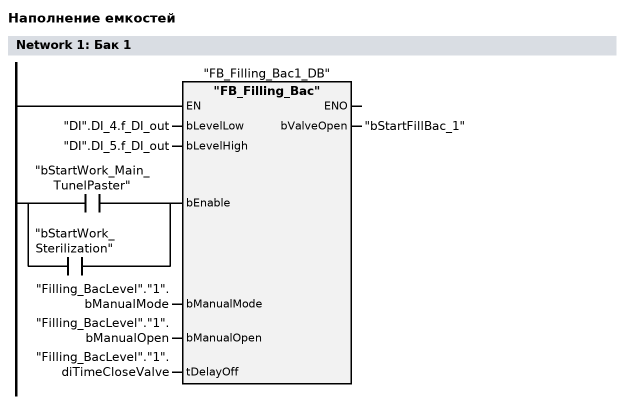
   RUNG wire#powerrail
      "FB_Filling_Bac1_DB"(bEnable := wire#w1, bLevelLow := "DI".DI_4.f_DI_out, bLevelHigh := "DI".DI_5.f_DI_out, bManualMode := "Filling_BacLevel"."1".bManualMode, bManualOpen := "Filling_BacLevel"."1".bManualOpen, tDelayOff := "Filling_BacLevel"."1".diTimeCloseValve, bValveOpen => "bStartFillBac_1")
   END_RUNG
   RUNG wire#powerrail
      Contact( "bStartWork_Main_TunelPaster" )
   END_RUNG wire#w1
   RUNG wire#powerrail
      Contact( "bStartWork_Sterilization" )
   END_RUNG wire#w1
   // the same network as SCL:
   "FB_Filling_Bac1_DB"(bLevelLow := "DI".DI_4.f_DI_out,   // "FB_Filling_Bac"
                        bLevelHigh := "DI".DI_5.f_DI_out,
                        bEnable := "bStartWork_Main_TunelPaster" OR "bStartWork_Sterilization",
                        bManualMode := "Filling_BacLevel"."1".bManualMode,
                        bManualOpen := "Filling_BacLevel"."1".bManualOpen,
                        tDelayOff := "Filling_BacLevel"."1".diTimeCloseValve,
                        bValveOpen => "bStartFillBac_1");
END_REGION
END_FUNCTION

FUNCTION "Все в Авто" : Void   // FC12, SCL
{ S7_Optimized_Access := 'TRUE' }
VERSION : 0.1
   VAR_TEMP
      fTrig_All_Auto : Bool;   // Фронт нажития кнопки все в авто
   END_VAR
BEGIN

   //Отлавливаем фронт нажатия клавиши все в авто
   "R_trig_All_Auto"(In:="bAllAuto",
                     Q=>#fTrig_All_Auto);

   //Сбрасываем все ручное в автоматический режим
   //
   IF #fTrig_All_Auto THEN

       //симуляция датчиков аналоговых
       "AI_DB".AI_1.bSimulate := FALSE;
       "AI_DB".AI_2.bSimulate := FALSE;
       "AI_DB".AI_3.bSimulate := FALSE;
       "AI_DB".AI_4.bSimulate := FALSE;
       "AI_DB".AI_5.bSimulate := FALSE;

       "AI_DB"."AI_4-20_1".bSimulate := FALSE;
       "AI_DB"."AI_4-20_2".bSimulate := FALSE;
       "AI_DB"."AI_4-20_3".bSimulate := FALSE;

       //Управление конвейером в ручном режиме
       "Conveyor".Conveyor_1.bManualMode := FALSE;
       "Conveyor".Conveyor_2.bManualMode := FALSE;
       "Conveyor".Conveyor_3.bManualMode := FALSE;
       "Conveyor".Conveyor_4.bManualMode := FALSE;

       //Управление баками наполнения
       "Filling_BacLevel"."1".bManualMode := FALSE;


       //Управление FV
       "FVs_o/p".FV_1.bManualMode := FALSE;
       "FVs_o/p".FV_2.bManualMode := FALSE;
       "FVs_o/p".FV_3.bManualMode := FALSE;


       //Управление Pumps
       "Pumps".Pump_1.bManualMode := FALSE;
       "Pumps".Pump_2.bManualMode := FALSE;
       "Pumps".Pump_3.bManualMode := FALSE;
       "Pumps".Pump_4.bManualMode := FALSE;
       "Pumps".Pump_5.bManualMode := FALSE;

       //Управление Vent
       "Vent".Vent_1.bManualMode := FALSE;

       //DI
       (*
       "DI".DI_0.bSimulation := FALSE;
       "DI".DI_1.bSimulation := FALSE;
       "DI".DI_2.bSimulation := FALSE;
       "DI".DI_3.bSimulation := FALSE;
       "DI".DI_4.bSimulation := FALSE;
       "DI".DI_5.bSimulation := FALSE;
       "DI".DI_6.bSimulation := FALSE;
       "DI".DI_7.bSimulation := FALSE;
       "DI".DI_8.bSimulation := FALSE;
       "DI".DI_9.bSimulation := FALSE;
       "DI".DI_10.bSimulation := FALSE;
       "DI".DI_11.bSimulation := FALSE;
       "DI".DI_12.bSimulation := FALSE;
       "DI".DI_13.bSimulation := FALSE;
       "DI".DI_14.bSimulation := FALSE;
       "DI".DI_15.bSimulation := FALSE;
       "DI".DI_16.bSimulation := FALSE;
       "DI".DI_17.bSimulation := FALSE;
       "DI".DI_18.bSimulation := FALSE;
       "DI".DI_19.bSimulation := FALSE;
       "DI".DI_20.bSimulation := FALSE;
       "DI".DI_21.bSimulation := FALSE;
       "DI".DI_22.bSimulation := FALSE;
       "DI".DI_23.bSimulation := FALSE;
       "DI".DI_24.bSimulation := FALSE;
       "DI".DI_25.bSimulation := FALSE;
       "DI".DI_26.bSimulation := FALSE;
       "DI".DI_27.bSimulation := FALSE;
       "DI".DI_28.bSimulation := FALSE;
       "DI".DI_29.bSimulation := FALSE;
      *)
   END_IF;
END_FUNCTION

FUNCTION "RestetAlarms" : Void   // FC13, SCL
{ S7_Optimized_Access := 'TRUE' }
VERSION : 0.1
BEGIN
   IF "bResetCommon" THEN
       //Сброс аварий насосов
       "Pumps".Pump_1.bresAlarm := TRUE;
       "Pumps".Pump_2.bresAlarm := TRUE;
       "Pumps".Pump_3.bresAlarm := TRUE;
       "Pumps".Pump_4.bresAlarm := TRUE;
       "Pumps".Pump_5.bresAlarm := TRUE;

       //Сброс аварий конвейера
       "Conveyor".Conveyor_1.bresAlarm := TRUE;
       "Conveyor".Conveyor_2.bresAlarm := TRUE;
       "Conveyor".Conveyor_3.bresAlarm := TRUE;
       "Conveyor".Conveyor_4.bresAlarm := TRUE;

       //Сброс аварий вентилятор
       "Vent".Vent_1.bresAlarm := TRUE;

       //Сброс аварий клапана
       "FVs_o/p".FV_1.bResetAlarm := TRUE;
       "FVs_o/p".FV_2.bResetAlarm := TRUE;
       "FVs_o/p".FV_3.bResetAlarm := TRUE;



   ELSE
       //Сброс аварий насосов
       "Pumps".Pump_1.bresAlarm := False;
       "Pumps".Pump_2.bresAlarm := False;
       "Pumps".Pump_3.bresAlarm := False;
       "Pumps".Pump_4.bresAlarm := False;
       "Pumps".Pump_5.bresAlarm := False;

       //Сброс аварий конвейера
       "Conveyor".Conveyor_1.bresAlarm := False;
       "Conveyor".Conveyor_2.bresAlarm := False;
       "Conveyor".Conveyor_3.bresAlarm := False;
       "Conveyor".Conveyor_4.bresAlarm := False;

       //Сброс аварий вентилятор
       "Vent".Vent_1.bresAlarm := FALSE;

       //Сброс аварий клапана
       "FVs_o/p".FV_1.bResetAlarm := False;
       "FVs_o/p".FV_2.bResetAlarm := False;
       "FVs_o/p".FV_3.bResetAlarm := False;


   END_IF;
END_FUNCTION

FUNCTION "Зоны Стерилизации_Контроль" : Void   // FC14, LAD
{ S7_Optimized_Access := 'TRUE' }
VERSION : 0.1
BEGIN

REGION Network 1: Зона 1
   // Зона 1
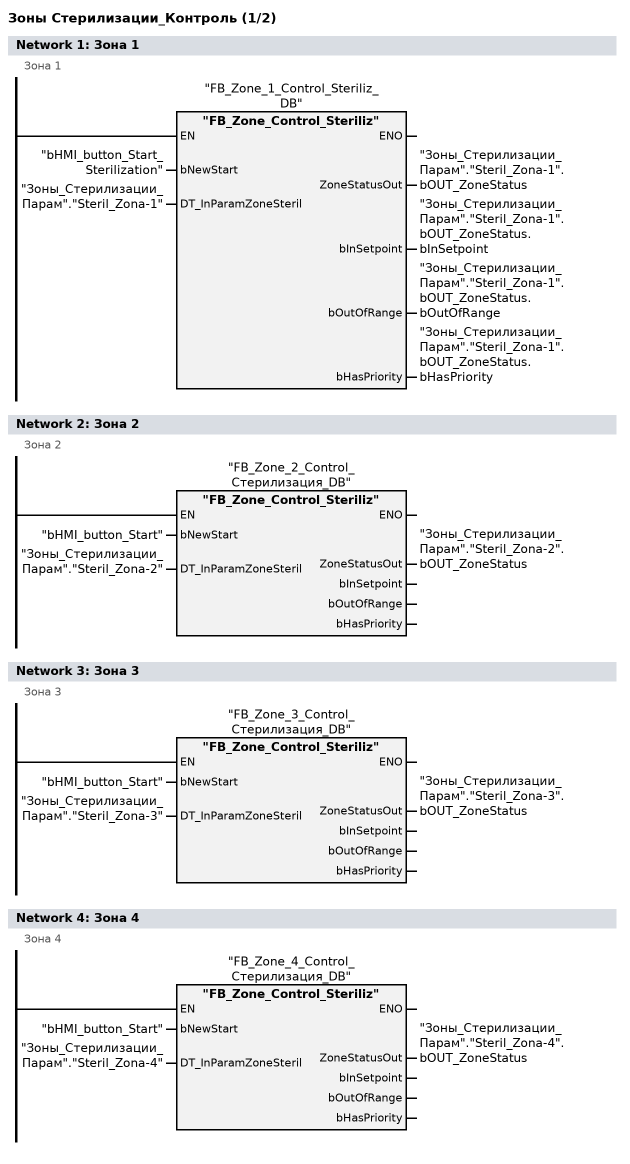
   RUNG wire#powerrail
      "FB_Zone_1_Control_Steriliz_DB"(bNewStart := "bHMI_button_Start_Sterilization", DT_InParamZoneSteril := "Зоны_Стерилизации_Парам"."Steril_Zona-1", ZoneStatusOut => "Зоны_Стерилизации_Парам"."Steril_Zona-1".bOUT_ZoneStatus, bInSetpoint => "Зоны_Стерилизации_Парам"."Steril_Zona-1".bOUT_ZoneStatus.bInSetpoint, bOutOfRange => "Зоны_Стерилизации_Парам"."Steril_Zona-1".bOUT_ZoneStatus.bOutOfRange, bHasPriority => "Зоны_Стерилизации_Парам"."Steril_Zona-1".bOUT_ZoneStatus.bHasPriority)
   END_RUNG
   // the same network as SCL:
   "FB_Zone_1_Control_Steriliz_DB"(bNewStart := "bHMI_button_Start_Sterilization",   // "FB_Zone_Control_Steriliz"
                           DT_InParamZoneSteril := "Зоны_Стерилизации_Парам"."Steril_Zona-1",
                           ZoneStatusOut => "Зоны_Стерилизации_Парам"."Steril_Zona-1".bOUT_ZoneStatus,
                           bInSetpoint => "Зоны_Стерилизации_Парам"."Steril_Zona-1".bOUT_ZoneStatus.bInSetpoint,
                           bOutOfRange => "Зоны_Стерилизации_Парам"."Steril_Zona-1".bOUT_ZoneStatus.bOutOfRange,
                           bHasPriority => "Зоны_Стерилизации_Парам"."Steril_Zona-1".bOUT_ZoneStatus.bHasPriority);
END_REGION

REGION Network 2: Зона 2
   // Зона 2
   RUNG wire#powerrail
      "FB_Zone_2_Control_Стерилизация_DB"(bNewStart := "bHMI_button_Start", DT_InParamZoneSteril := "Зоны_Стерилизации_Парам"."Steril_Zona-2", ZoneStatusOut => "Зоны_Стерилизации_Парам"."Steril_Zona-2".bOUT_ZoneStatus, bInSetpoint =>, bOutOfRange =>, bHasPriority =>)
   END_RUNG
   // the same network as SCL:
   "FB_Zone_2_Control_Стерилизация_DB"(bNewStart := "bHMI_button_Start",   // "FB_Zone_Control_Steriliz"
                           DT_InParamZoneSteril := "Зоны_Стерилизации_Парам"."Steril_Zona-2",
                           ZoneStatusOut => "Зоны_Стерилизации_Парам"."Steril_Zona-2".bOUT_ZoneStatus);
END_REGION

REGION Network 3: Зона 3
   // Зона 3
   RUNG wire#powerrail
      "FB_Zone_3_Control_Стерилизация_DB"(bNewStart := "bHMI_button_Start", DT_InParamZoneSteril := "Зоны_Стерилизации_Парам"."Steril_Zona-3", ZoneStatusOut => "Зоны_Стерилизации_Парам"."Steril_Zona-3".bOUT_ZoneStatus, bInSetpoint =>, bOutOfRange =>, bHasPriority =>)
   END_RUNG
   // the same network as SCL:
   "FB_Zone_3_Control_Стерилизация_DB"(bNewStart := "bHMI_button_Start",   // "FB_Zone_Control_Steriliz"
                           DT_InParamZoneSteril := "Зоны_Стерилизации_Парам"."Steril_Zona-3",
                           ZoneStatusOut => "Зоны_Стерилизации_Парам"."Steril_Zona-3".bOUT_ZoneStatus);
END_REGION

REGION Network 4: Зона 4
   // Зона 4
   RUNG wire#powerrail
      "FB_Zone_4_Control_Стерилизация_DB"(bNewStart := "bHMI_button_Start", DT_InParamZoneSteril := "Зоны_Стерилизации_Парам"."Steril_Zona-4", ZoneStatusOut => "Зоны_Стерилизации_Парам"."Steril_Zona-4".bOUT_ZoneStatus, bInSetpoint =>, bOutOfRange =>, bHasPriority =>)
   END_RUNG
   // the same network as SCL:
   "FB_Zone_4_Control_Стерилизация_DB"(bNewStart := "bHMI_button_Start",   // "FB_Zone_Control_Steriliz"
                           DT_InParamZoneSteril := "Зоны_Стерилизации_Парам"."Steril_Zona-4",
                           ZoneStatusOut => "Зоны_Стерилизации_Парам"."Steril_Zona-4".bOUT_ZoneStatus);
END_REGION

REGION Network 5: Зона 5
   // Зона 5
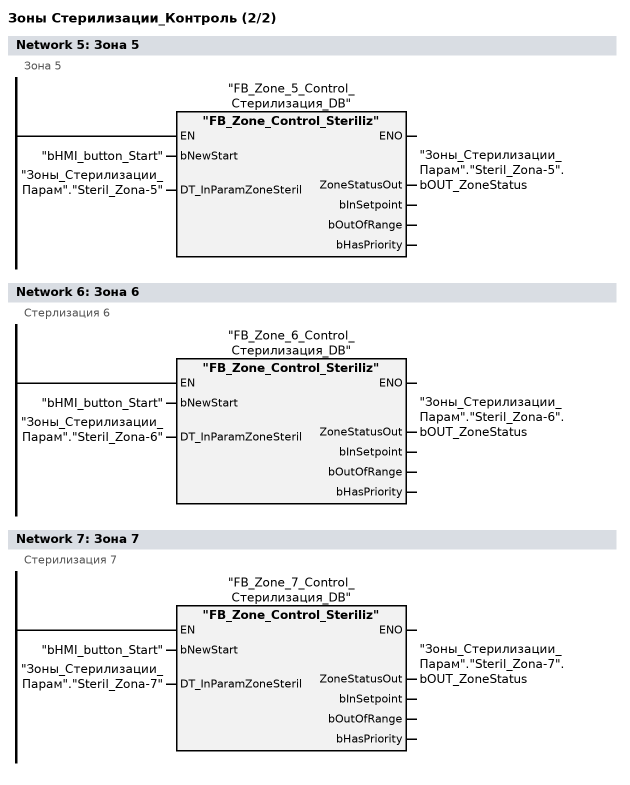
   RUNG wire#powerrail
      "FB_Zone_5_Control_Стерилизация_DB"(bNewStart := "bHMI_button_Start", DT_InParamZoneSteril := "Зоны_Стерилизации_Парам"."Steril_Zona-5", ZoneStatusOut => "Зоны_Стерилизации_Парам"."Steril_Zona-5".bOUT_ZoneStatus, bInSetpoint =>, bOutOfRange =>, bHasPriority =>)
   END_RUNG
   // the same network as SCL:
   "FB_Zone_5_Control_Стерилизация_DB"(bNewStart := "bHMI_button_Start",   // "FB_Zone_Control_Steriliz"
                           DT_InParamZoneSteril := "Зоны_Стерилизации_Парам"."Steril_Zona-5",
                           ZoneStatusOut => "Зоны_Стерилизации_Парам"."Steril_Zona-5".bOUT_ZoneStatus);
END_REGION

REGION Network 6: Зона 6
   // Стерлизация 6
   RUNG wire#powerrail
      "FB_Zone_6_Control_Стерилизация_DB"(bNewStart := "bHMI_button_Start", DT_InParamZoneSteril := "Зоны_Стерилизации_Парам"."Steril_Zona-6", ZoneStatusOut => "Зоны_Стерилизации_Парам"."Steril_Zona-6".bOUT_ZoneStatus, bInSetpoint =>, bOutOfRange =>, bHasPriority =>)
   END_RUNG
   // the same network as SCL:
   "FB_Zone_6_Control_Стерилизация_DB"(bNewStart := "bHMI_button_Start",   // "FB_Zone_Control_Steriliz"
                           DT_InParamZoneSteril := "Зоны_Стерилизации_Парам"."Steril_Zona-6",
                           ZoneStatusOut => "Зоны_Стерилизации_Парам"."Steril_Zona-6".bOUT_ZoneStatus);
END_REGION

REGION Network 7: Зона 7
   // Стерилизация 7
   RUNG wire#powerrail
      "FB_Zone_7_Control_Стерилизация_DB"(bNewStart := "bHMI_button_Start", DT_InParamZoneSteril := "Зоны_Стерилизации_Парам"."Steril_Zona-7", ZoneStatusOut => "Зоны_Стерилизации_Парам"."Steril_Zona-7".bOUT_ZoneStatus, bInSetpoint =>, bOutOfRange =>, bHasPriority =>)
   END_RUNG
   // the same network as SCL:
   "FB_Zone_7_Control_Стерилизация_DB"(bNewStart := "bHMI_button_Start",   // "FB_Zone_Control_Steriliz"
                           DT_InParamZoneSteril := "Зоны_Стерилизации_Парам"."Steril_Zona-7",
                           ZoneStatusOut => "Зоны_Стерилизации_Парам"."Steril_Zona-7".bOUT_ZoneStatus);
END_REGION

REGION Network 8 (SCL): Соответствие выхода с датчика температур с входом для темп зоны
   "Зоны_Стерилизации_Парам"."Steril_Zona-1".rTemp := "AI_DB".AI_1.rAI_Value;
   "Зоны_Стерилизации_Парам"."Steril_Zona-2".rTemp := "AI_DB".AI_2.rAI_Value;
   "Зоны_Стерилизации_Парам"."Steril_Zona-3".rTemp := "AI_DB".AI_3.rAI_Value;
   "Зоны_Стерилизации_Парам"."Steril_Zona-4".rTemp := "AI_DB".AI_4.rAI_Value;
   "Зоны_Стерилизации_Парам"."Steril_Zona-5".rTemp := "AI_DB".AI_5.rAI_Value;
   "Зоны_Стерилизации_Парам"."Steril_Zona-6".rTemp := "AI_DB".AI_6.rAI_Value;
   "Зоны_Стерилизации_Парам"."Steril_Zona-7".rTemp := "AI_DB".AI_7.rAI_Value;
END_REGION
END_FUNCTION

FUNCTION "PressControl" : Void   // FC15, SCL
{ S7_Optimized_Access := 'TRUE' }
VERSION : 0.1
BEGIN

   // ---------------Присваиваем значения переменным------------------
   // 
   "Control_Press_DB".PressWater.rInPress := "AI_DB"."AI_4-20_1".rAI_Value;
   "Control_Press_DB".PressSteam.rInPress := "AI_DB"."AI_4-20_2".rAI_Value;
   "Control_Press_DB".PressGlikol.rInPress := "AI_DB"."AI_4-20_3".rAI_Value;


   //Давление ПАРА..................................................

   "FB_Press_Controll_Steam_DB"("Control_Press_DB".PressSteam);


   //Давление Воды..................................................

   "FB_Press_Controll_Water_DB"("Control_Press_DB".PressWater);


   //Давление Гликоля..................................................

   "FB_Press_Controll_Glikol_DB"("Control_Press_DB".PressGlikol);
END_FUNCTION

ORGANIZATION_BLOCK "Main"   // OB1, LAD, ProgramCycle
TITLE = "Основкая программа"
{ S7_Optimized_Access := 'TRUE' }
VERSION : 0.1
   VAR_TEMP
      Test1 : Bool;
   END_VAR
BEGIN

REGION Network 1: Аварии
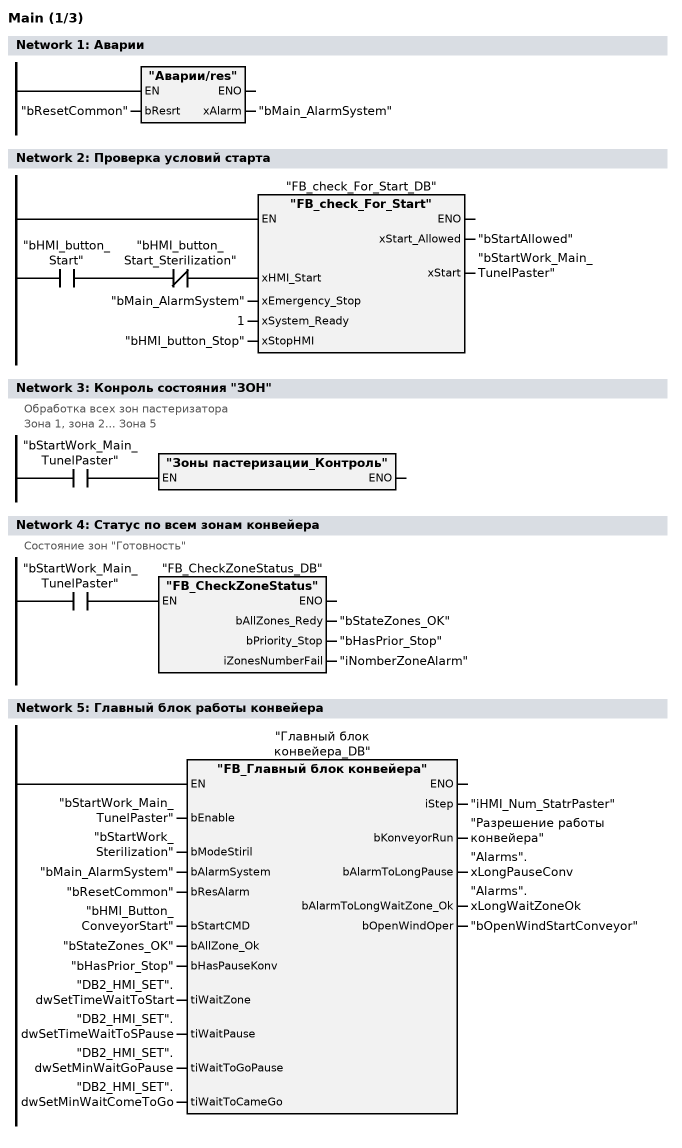
   RUNG wire#powerrail
      "Аварии/res"(bResrt := "bResetCommon", xAlarm => "bMain_AlarmSystem")
   END_RUNG
   // the same network as SCL:
   "Аварии/res"(bResrt := "bResetCommon", xAlarm => "bMain_AlarmSystem");
END_REGION

REGION Network 2: Проверка условий старта
   RUNG wire#powerrail
      "FB_check_For_Start_DB"(xHMI_Start := wire#w1, xEmergency_Stop := "bMain_AlarmSystem", xSystem_Ready := 1, xStopHMI := "bHMI_button_Stop", xStart_Allowed => "bStartAllowed", xStart => "bStartWork_Main_TunelPaster")
   END_RUNG
   RUNG wire#powerrail
      Contact( "bHMI_button_Start" )
      I_Contact( "bHMI_button_Start_Sterilization" )
   END_RUNG wire#w1
   // the same network as SCL:
   "FB_check_For_Start_DB"(xHMI_Start := "bHMI_button_Start" AND NOT "bHMI_button_Start_Sterilization",   // "FB_check_For_Start"
                           xEmergency_Stop := "bMain_AlarmSystem",
                           xSystem_Ready := 1,
                           xStopHMI := "bHMI_button_Stop",
                           xStart_Allowed => "bStartAllowed",
                           xStart => "bStartWork_Main_TunelPaster");
END_REGION

REGION Network 3: Конроль состояния "ЗОН"
   // Обработка всех зон пастеризатора
   // Зона 1, зона 2... Зона 5
   RUNG wire#powerrail
      Contact( "bStartWork_Main_TunelPaster" )
      "Зоны пастеризации_Контроль"()
   END_RUNG
   // the same network as SCL:
   IF "bStartWork_Main_TunelPaster" THEN "Зоны пастеризации_Контроль"(); END_IF;
END_REGION

REGION Network 4: Статус по всем зонам конвейера
   // Состояние зон "Готовность"
   RUNG wire#powerrail
      Contact( "bStartWork_Main_TunelPaster" )
      "FB_CheckZoneStatus_DB"(bAllZones_Redy => "bStateZones_OK", bPriority_Stop => "bHasPrior_Stop", iZonesNumberFail => "iNomberZoneAlarm")
   END_RUNG
   // the same network as SCL:
   IF "bStartWork_Main_TunelPaster" THEN
       "FB_CheckZoneStatus_DB"(bAllZones_Redy => "bStateZones_OK",   // "FB_CheckZoneStatus"
                               bPriority_Stop => "bHasPrior_Stop",
                               iZonesNumberFail => "iNomberZoneAlarm");
   END_IF;
END_REGION

REGION Network 5: Главный блок работы конвейера
   RUNG wire#powerrail
      "Главный блок конвейера_DB"(bEnable := "bStartWork_Main_TunelPaster", bModeStiril := "bStartWork_Sterilization", bAlarmSystem := "bMain_AlarmSystem", bResAlarm := "bResetCommon", bStartCMD := "bHMI_Button_ConveyorStart", bAllZone_Ok := "bStateZones_OK", bHasPauseKonv := "bHasPrior_Stop", tiWaitZone := "DB2_HMI_SET".dwSetTimeWaitToStart, tiWaitPause := "DB2_HMI_SET".dwSetTimeWaitToSPause, tiWaitToGoPause := "DB2_HMI_SET".dwSetMinWaitGoPause, tiWaitToCameGo := "DB2_HMI_SET".dwSetMinWaitComeToGo, iStep => "iHMI_Num_StatrPaster", bKonveyorRun => "Разрешение работы конвейера", bAlarmToLongPause => "Alarms".xLongPauseConv, bAlarmToLongWaitZone_Ok => "Alarms".xLongWaitZoneOk, bOpenWindOper => "bOpenWindStartConveyor")
   END_RUNG
   // the same network as SCL:
   "Главный блок конвейера_DB"(bEnable := "bStartWork_Main_TunelPaster",   // "FB_Главный блок конвейера"
                           bModeStiril := "bStartWork_Sterilization",
                           bAlarmSystem := "bMain_AlarmSystem",
                           bResAlarm := "bResetCommon",
                           bStartCMD := "bHMI_Button_ConveyorStart",
                           bAllZone_Ok := "bStateZones_OK",
                           bHasPauseKonv := "bHasPrior_Stop",
                           tiWaitZone := "DB2_HMI_SET".dwSetTimeWaitToStart,
                           tiWaitPause := "DB2_HMI_SET".dwSetTimeWaitToSPause,
                           tiWaitToGoPause := "DB2_HMI_SET".dwSetMinWaitGoPause,
                           tiWaitToCameGo := "DB2_HMI_SET".dwSetMinWaitComeToGo,
                           iStep => "iHMI_Num_StatrPaster",
                           bKonveyorRun => "Разрешение работы конвейера",
                           bAlarmToLongPause => "Alarms".xLongPauseConv,
                           bAlarmToLongWaitZone_Ok => "Alarms".xLongWaitZoneOk,
                           bOpenWindOper => "bOpenWindStartConveyor");
END_REGION

REGION Network 6: Расчет PE и скорости конвейера
